LIN {X 0,Y 340.685,Z 308.673,A -85,B 0,C 180,E1 -14072.436,E2 -14072.436} C_VEL
LIN {X 0,Y 340.717,Z 308.669,A -85,B 0,C 180,E1 -14075.279,E2 -14075.279} C_VEL
LIN {X 0,Y 340.751,Z 308.84,A -85,B 0,C 180,E1 -14077.57,E2 -14077.57} C_VEL
LIN {X 0,Y 342.607,Z 316.882,A -85,B 0,C 180,E1 -14081.028,E2 -14081.028} C_VEL
LIN {X 0,Y 344.616,Z 325.417,A -85,B 0,C 180,E1 -14084.457,E2 -14084.457} C_VEL
LIN {X 0,Y 346.876,Z 334.938,A -85,B 0,C 180,E1 -14088.041,E2 -14088.041} C_VEL
LIN {X 0,Y 349.374,Z 345.213,A -85,B 0,C 180,E1 -14091.676,E2 -14091.676} C_VEL
LIN {X 0,Y 349.814,Z 347.163,A -85,B 0,C 180,E1 -14092.337,E2 -14092.337} C_VEL
LIN {X 0,Y 348.93,Z 352.343,A -85,B 0,C 180,E1 -14093.935,E2 -14093.935} C_VEL
LIN {X 0,Y 346.318,Z 365.305,A -85,B 0,C 180,E1 -14097.812,E2 -14097.812} C_VEL
LIN {X 0,Y 345.144,Z 372.439,A -85,B 0,C 180,E1 -14099.865,E2 -14099.865} C_VEL
LIN {X 0,Y 345.357,Z 374.641,A -85,B 0,C 180,E1 -14100,E2 -14100} C_VEL
LIN {X 0,Y 349.581,Z 396.16,A -85,B 0,C 180,E1 -14100.94,E2 -14100.94} C_VEL
LIN {X 0,Y 351.629,Z 411.603,A -85,B 0,C 180,E1 -14101.761,E2 -14101.761} C_VEL
LIN {X 0,Y 353.04,Z 426.596,A -85,B 0,C 180,E1 -14102.751,E2 -14102.751} C_VEL
LIN {X 0,Y 353.156,Z 435.408,A -85,B 0,C 180,E1 -14103.401,E2 -14103.401} C_VEL
LIN {X 0,Y 351.443,Z 448.562,A -85,B 0,C 180,E1 -14104.412,E2 -14104.412} C_VEL
LIN {X 0,Y 349.424,Z 461.614,A -85,B 0,C 180,E1 -14105.65,E2 -14105.65} C_VEL
LIN {X 0,Y 347.416,Z 473.933,A -85,B 0,C 180,E1 -14107.082,E2 -14107.082} C_VEL
LIN {X 0,Y 345.407,Z 486.223,A -85,B 0,C 180,E1 -14108.829,E2 -14108.829} C_VEL
LIN {X 0,Y 343.692,Z 496.83,A -85,B 0,C 180,E1 -14110.646,E2 -14110.646} C_VEL
LIN {X 0,Y 342.121,Z 506.665,A -85,B 0,C 180,E1 -14112.671,E2 -14112.671} C_VEL
LIN {X 0,Y 340.951,Z 515.073,A -85,B 0,C 180,E1 -14114.763,E2 -14114.763} C_VEL
LIN {X 0,Y 340.104,Z 522.05,A -85,B 0,C 180,E1 -14116.862,E2 -14116.862} C_VEL
LIN {X 0,Y 339.576,Z 528.54,A -85,B 0,C 180,E1 -14119.265,E2 -14119.265} C_VEL
LIN {X 0,Y 339.406,Z 533.572,A -85,B 0,C 180,E1 -14121.666,E2 -14121.666} C_VEL
LIN {X 0,Y 339.511,Z 537.273,A -85,B 0,C 180,E1 -14124.059,E2 -14124.059} C_VEL
LIN {X 0,Y 339.588,Z 539.71,A -85,B 0,C 180,E1 -14126.441,E2 -14126.441} C_VEL
LIN {X 0,Y 339.726,Z 540.943,A -85,B 0,C 180,E1 -14128.815,E2 -14128.815} C_VEL
LIN {X 0,Y 339.728,Z 540.942,A -85,B 0,C 180,E1 -14131.186,E2 -14131.186} C_VEL
LIN {X 0,Y 339.614,Z 539.708,A -85,B 0,C 180,E1 -14133.56,E2 -14133.56} C_VEL
LIN {X 0,Y 339.55,Z 537.267,A -85,B 0,C 180,E1 -14135.94,E2 -14135.94} C_VEL
LIN {X 0,Y 339.48,Z 533.556,A -85,B 0,C 180,E1 -14138.333,E2 -14138.333} C_VEL
LIN {X 0,Y 339.601,Z 528.509,A -85,B 0,C 180,E1 -14140.735,E2 -14140.735} C_VEL
LIN {X 0,Y 340.154,Z 522.02,A -85,B 0,C 180,E1 -14143.137,E2 -14143.137} C_VEL
LIN {X 0,Y 340.959,Z 515.032,A -85,B 0,C 180,E1 -14145.237,E2 -14145.237} C_VEL
LIN {X 0,Y 342.106,Z 506.607,A -85,B 0,C 180,E1 -14147.331,E2 -14147.331} C_VEL
LIN {X 0,Y 343.781,Z 496.672,A -85,B 0,C 180,E1 -14149.369,E2 -14149.369} C_VEL
LIN {X 0,Y 345.421,Z 486.141,A -85,B 0,C 180,E1 -14151.171,E2 -14151.171} C_VEL
LIN {X 0,Y 347.463,Z 473.824,A -85,B 0,C 180,E1 -14152.915,E2 -14152.915} C_VEL
LIN {X 0,Y 349.475,Z 461.488,A -85,B 0,C 180,E1 -14154.347,E2 -14154.347} C_VEL
LIN {X 0,Y 351.409,Z 448.341,A -85,B 0,C 180,E1 -14155.598,E2 -14155.598} C_VEL
LIN {X 0,Y 353.949,Z 433.264,A -85,B 0,C 180,E1 -14157.014,E2 -14157.014} C_VEL
LIN {X 0,Y 354.679,Z 418.66,A -85,B 0,C 180,E1 -14158.396,E2 -14158.396} C_VEL
LIN {X 0,Y 354.576,Z 406.998,A -85,B 0,C 180,E1 -14159.443,E2 -14159.443} C_VEL
LIN {X 0,Y 353.206,Z 394.587,A -85,B 0,C 180,E1 -14160.595,E2 -14160.595} C_VEL
LIN {X 0,Y 350.848,Z 381.951,A -85,B 0,C 180,E1 -14161.846,E2 -14161.846} C_VEL
LIN {X 0,Y 349.008,Z 374.393,A -85,B 0,C 180,E1 -14162.655,E2 -14162.655} C_VEL
LIN {X 0,Y 348.091,Z 370.111,A -85,B 0,C 180,E1 -14163.12,E2 -14163.12} C_VEL
LIN {X 0,Y 350.836,Z 361.608,A -85,B 0,C 180,E1 -14166.225,E2 -14166.225} C_VEL
LIN {X 0,Y 352.145,Z 358.36,A -85,B 0,C 180,E1 -14167.496,E2 -14167.496} C_VEL
LIN {X 0,Y 352.45,Z 356.806,A -85,B 0,C 180,E1 -14168.182,E2 -14168.182} C_VEL
LIN {X 0,Y 351.555,Z 352.589,A -85,B 0,C 180,E1 -14170.565,E2 -14170.565} C_VEL
LIN {X 0,Y 350.19,Z 348.108,A -85,B 0,C 180,E1 -14173.74,E2 -14173.74} C_VEL
LIN {X 0,Y 349.169,Z 344.785,A -85,B 0,C 180,E1 -14176.816,E2 -14176.816} C_VEL
LIN {X 0,Y 348.17,Z 342.313,A -85,B 0,C 180,E1 -14180.09,E2 -14180.09} C_VEL
LIN {X 0,Y 347.502,Z 341.045,A -85,B 0,C 180,E1 -14182.647,E2 -14182.647} C_VEL
LIN {X 0,Y 346.648,Z 340.315,A -85,B 0,C 180,E1 -14185.412,E2 -14185.412} C_VEL
LIN {X 0,Y 345.766,Z 340.093,A -85,B 0,C 180,E1 -14188.616,E2 -14188.616} C_VEL
LIN {X 0,Y 345.131,Z 340.385,A -85,B 0,C 180,E1 -14191.526,E2 -14191.526} C_VEL
LIN {X 0,Y 346.63,Z 343.275,A -85,B 0,C 180,E1 -14192.204,E2 -14192.204} C_VEL
LIN {X 0,Y 350.286,Z 348.385,A -85,B 0,C 180,E1 -14193.557,E2 -14193.557} C_VEL
LIN {X 0,Y 355.192,Z 357.489,A -85,B 0,C 180,E1 -14195.531,E2 -14195.531} C_VEL
LIN {X 0,Y 358.558,Z 365.842,A -85,B 0,C 180,E1 -14197.108,E2 -14197.108} C_VEL
LIN {X 0,Y 359.707,Z 369.419,A -85,B 0,C 180,E1 -14197.752,E2 -14197.752} C_VEL
LIN {X 0,Y 357.203,Z 382.897,A -85,B 0,C 180,E1 -14199.259,E2 -14199.259} C_VEL
LIN {X 0,Y 354.992,Z 392.974,A -85,B 0,C 180,E1 -14200.634,E2 -14200.634} C_VEL
LIN {X 0,Y 352.597,Z 403.108,A -85,B 0,C 180,E1 -14202.304,E2 -14202.304} C_VEL
LIN {X 0,Y 350.494,Z 411.648,A -85,B 0,C 180,E1 -14204.026,E2 -14204.026} C_VEL
LIN {X 0,Y 348.293,Z 419.501,A -85,B 0,C 180,E1 -14205.987,E2 -14205.987} C_VEL
LIN {X 0,Y 346.67,Z 425.084,A -85,B 0,C 180,E1 -14207.71,E2 -14207.71} C_VEL
LIN {X 0,Y 345.306,Z 429.544,A -85,B 0,C 180,E1 -14209.445,E2 -14209.445} C_VEL
LIN {X 0,Y 343.702,Z 434.016,A -85,B 0,C 180,E1 -14211.771,E2 -14211.771} C_VEL
LIN {X 0,Y 343.116,Z 435.597,A -85,B 0,C 180,E1 -14212.941,E2 -14212.941} C_VEL
LIN {X 0,Y 342.313,Z 437.544,A -85,B 0,C 180,E1 -14215.289,E2 -14215.289} C_VEL
LIN {X 0,Y 341.557,Z 438.025,A -85,B 0,C 180,E1 -14217.642,E2 -14217.642} C_VEL
LIN {X 0,Y 341.362,Z 437.648,A -85,B 0,C 180,E1 -14218.82,E2 -14218.82} C_VEL
LIN {X 0,Y 341.018,Z 436.906,A -85,B 0,C 180,E1 -14220,E2 -14220} C_VEL
LIN {X 0,Y 340.978,Z 435.738,A -85,B 0,C 180,E1 -14221.181,E2 -14221.181} C_VEL
LIN {X 0,Y 340.851,Z 434.198,A -85,B 0,C 180,E1 -14222.364,E2 -14222.364} C_VEL
LIN {X 0,Y 340.813,Z 431.07,A -85,B 0,C 180,E1 -14224.139,E2 -14224.139} C_VEL
LIN {X 0,Y 341.181,Z 426.928,A -85,B 0,C 180,E1 -14225.912,E2 -14225.912} C_VEL
LIN {X 0,Y 341.536,Z 421.737,A -85,B 0,C 180,E1 -14227.687,E2 -14227.687} C_VEL
LIN {X 0,Y 342.068,Z 414.154,A -85,B 0,C 180,E1 -14229.759,E2 -14229.759} C_VEL
LIN {X 0,Y 342.657,Z 406.099,A -85,B 0,C 180,E1 -14231.536,E2 -14231.536} C_VEL
LIN {X 0,Y 343.362,Z 396.351,A -85,B 0,C 180,E1 -14233.313,E2 -14233.313} C_VEL
LIN {X 0,Y 344.291,Z 385.473,A -85,B 0,C 180,E1 -14234.935,E2 -14234.935} C_VEL
LIN {X 0,Y 345.287,Z 373.449,A -85,B 0,C 180,E1 -14236.404,E2 -14236.404} C_VEL
LIN {X 0,Y 346.141,Z 361.256,A -85,B 0,C 180,E1 -14237.624,E2 -14237.624} C_VEL
LIN {X 0,Y 346.99,Z 348.049,A -85,B 0,C 180,E1 -14238.679,E2 -14238.679} C_VEL
LIN {X 0,Y 343.823,Z 334.91,A -85,B 0,C 180,E1 -14239.681,E2 -14239.681} C_VEL
LIN {X 0,Y 340.174,Z 320.362,A -85,B 0,C 180,E1 -14240.562,E2 -14240.562} C_VEL
LIN {X 0,Y 340.178,Z 316.024,A -85,B 0,C 180,E1 -14244.627,E2 -14244.627} C_VEL
LIN {X 0,Y 340.19,Z 312.178,A -85,B 0,C 180,E1 -14248.37,E2 -14248.37} C_VEL
LIN {X 0,Y 340.199,Z 309.423,A -85,B 0,C 180,E1 -14251.095,E2 -14251.095} C_VEL
LIN {X 0,Y 340.306,Z 308.722,A -85,B 0,C 180,E1 -14252.477,E2 -14252.477} C_VEL
LIN {X 0,Y 340.556,Z 308.69,A -85,B 0,C 180,E1 -14255.298,E2 -14255.298} C_VEL
LIN {X 0,Y 340.705,Z 308.671,A -85,B 0,C 180,E1 -14258.384,E2 -14258.384} C_VEL
LIN {X 0,Y 340.701,Z 308.665,A -85,B 0,C 180,E1 -14262.045,E2 -14262.045} C_VEL
LIN {X 0,Y 340.707,Z 308.817,A -85,B 0,C 180,E1 -14263.132,E2 -14263.132} C_VEL
LIN {X 0,Y 341.39,Z 312.413,A -85,B 0,C 180,E1 -14266.098,E2 -14266.098} C_VEL
LIN {X 0,Y 341.716,Z 315.809,A -85,B 0,C 180,E1 -14268.842,E2 -14268.842} C_VEL
LIN {X 0,Y 341.73,Z 319.739,A -85,B 0,C 180,E1 -14271.904,E2 -14271.904} C_VEL
LIN {X 0,Y 341.66,Z 324.36,A -85,B 0,C 180,E1 -14275.367,E2 -14275.367} C_VEL
LIN {X 0,Y 341.617,Z 329.636,A -85,B 0,C 180,E1 -14279.048,E2 -14279.048} C_VEL
LIN {X 0,Y 341.643,Z 330.583,A -85,B 0,C 180,E1 -14279.625,E2 -14279.625} C_VEL
LIN {X 0,Y 343.082,Z 333.899,A -85,B 0,C 180,E1 -14279.849,E2 -14279.849} C_VEL
LIN {X 0,Y 349.127,Z 348.085,A -85,B 0,C 180,E1 -14280.902,E2 -14280.902} C_VEL
LIN {X 0,Y 354.05,Z 362.001,A -85,B 0,C 180,E1 -14282.041,E2 -14282.041} C_VEL
LIN {X 0,Y 356.741,Z 371.631,A -85,B 0,C 180,E1 -14282.881,E2 -14282.881} C_VEL
LIN {X 0,Y 355.481,Z 385.325,A -85,B 0,C 180,E1 -14283.838,E2 -14283.838} C_VEL
LIN {X 0,Y 353.788,Z 399.027,A -85,B 0,C 180,E1 -14285.03,E2 -14285.03} C_VEL
LIN {X 0,Y 351.753,Z 412.252,A -85,B 0,C 180,E1 -14286.447,E2 -14286.447} C_VEL
LIN {X 0,Y 349.877,Z 424.229,A -85,B 0,C 180,E1 -14288.03,E2 -14288.03} C_VEL
LIN {X 0,Y 347.873,Z 435.957,A -85,B 0,C 180,E1 -14289.913,E2 -14289.913} C_VEL
LIN {X 0,Y 346.162,Z 445.017,A -85,B 0,C 180,E1 -14291.658,E2 -14291.658} C_VEL
LIN {X 0,Y 344.321,Z 454.308,A -85,B 0,C 180,E1 -14293.804,E2 -14293.804} C_VEL
LIN {X 0,Y 343.032,Z 461.257,A -85,B 0,C 180,E1 -14295.767,E2 -14295.767} C_VEL
LIN {X 0,Y 341.82,Z 468.102,A -85,B 0,C 180,E1 -14298.135,E2 -14298.135} C_VEL
LIN {X 0,Y 340.917,Z 473.474,A -85,B 0,C 180,E1 -14300.507,E2 -14300.507} C_VEL
LIN {X 0,Y 340.273,Z 477.532,A -85,B 0,C 180,E1 -14302.881,E2 -14302.881} C_VEL
LIN {X 0,Y 340.001,Z 480.366,A -85,B 0,C 180,E1 -14305.257,E2 -14305.257} C_VEL
LIN {X 0,Y 339.76,Z 482.072,A -85,B 0,C 180,E1 -14307.629,E2 -14307.629} C_VEL
LIN {X 0,Y 339.624,Z 482.668,A -85,B 0,C 180,E1 -14310,E2 -14310} C_VEL
LIN {X 0,Y 339.755,Z 482.11,A -85,B 0,C 180,E1 -14312.371,E2 -14312.371} C_VEL
LIN {X 0,Y 339.998,Z 480.455,A -85,B 0,C 180,E1 -14314.743,E2 -14314.743} C_VEL
LIN {X 0,Y 340.272,Z 477.68,A -85,B 0,C 180,E1 -14317.118,E2 -14317.118} C_VEL
LIN {X 0,Y 340.909,Z 473.685,A -85,B 0,C 180,E1 -14319.493,E2 -14319.493} C_VEL
LIN {X 0,Y 341.793,Z 468.373,A -85,B 0,C 180,E1 -14321.866,E2 -14321.866} C_VEL
LIN {X 0,Y 343.01,Z 461.588,A -85,B 0,C 180,E1 -14324.233,E2 -14324.233} C_VEL
LIN {X 0,Y 344.226,Z 454.918,A -85,B 0,C 180,E1 -14326.142,E2 -14326.142} C_VEL
LIN {X 0,Y 346.053,Z 445.516,A -85,B 0,C 180,E1 -14328.348,E2 -14328.348} C_VEL
LIN {X 0,Y 348.106,Z 434.858,A -85,B 0,C 180,E1 -14330.381,E2 -14330.381} C_VEL
LIN {X 0,Y 349.849,Z 423.919,A -85,B 0,C 180,E1 -14332.127,E2 -14332.127} C_VEL
LIN {X 0,Y 351.938,Z 411.859,A -85,B 0,C 180,E1 -14333.696,E2 -14333.696} C_VEL
LIN {X 0,Y 353.85,Z 398.537,A -85,B 0,C 180,E1 -14335.121,E2 -14335.121} C_VEL
LIN {X 0,Y 355.533,Z 384.643,A -85,B 0,C 180,E1 -14336.32,E2 -14336.32} C_VEL
LIN {X 0,Y 356.766,Z 372.504,A -85,B 0,C 180,E1 -14337.161,E2 -14337.161} C_VEL
LIN {X 0,Y 355.958,Z 368.246,A -85,B 0,C 180,E1 -14337.515,E2 -14337.515} C_VEL
LIN {X 0,Y 351.475,Z 354.305,A -85,B 0,C 180,E1 -14338.709,E2 -14338.709} C_VEL
LIN {X 0,Y 345.813,Z 339.855,A -85,B 0,C 180,E1 -14339.821,E2 -14339.821} C_VEL
LIN {X 0,Y 341.718,Z 330.796,A -85,B 0,C 180,E1 -14340.473,E2 -14340.473} C_VEL
LIN {X 0,Y 341.639,Z 330.42,A -85,B 0,C 180,E1 -14340.544,E2 -14340.544} C_VEL
LIN {X 0,Y 341.624,Z 325.783,A -85,B 0,C 180,E1 -14343.742,E2 -14343.742} C_VEL
LIN {X 0,Y 341.659,Z 322.309,A -85,B 0,C 180,E1 -14346.3,E2 -14346.3} C_VEL
LIN {X 0,Y 341.072,Z 321.186,A -85,B 0,C 180,E1 -14347.266,E2 -14347.266} C_VEL
LIN {X 0,Y 338.315,Z 319.77,A -85,B 0,C 180,E1 -14348.851,E2 -14348.851} C_VEL
LIN {X 0,Y 335.921,Z 318.68,A -85,B 0,C 180,E1 -14350.136,E2 -14350.136} C_VEL
LIN {X 0,Y 334.857,Z 317.669,A -85,B 0,C 180,E1 -14351.124,E2 -14351.124} C_VEL
LIN {X 0,Y 334.753,Z 317.262,A -85,B 0,C 180,E1 -14351.456,E2 -14351.456} C_VEL
LIN {X 0,Y 334.404,Z 313.699,A -85,B 0,C 180,E1 -14354.393,E2 -14354.393} C_VEL
LIN {X 0,Y 333.652,Z 309.552,A -85,B 0,C 180,E1 -14357.824,E2 -14357.824} C_VEL
LIN {X 0,Y 333.652,Z 309.545,A -85,B 0,C 180,E1 -14361.202,E2 -14361.202} C_VEL
LIN {X 0,Y 333.676,Z 309.541,A -85,B 0,C 180,E1 -14363.861,E2 -14363.861} C_VEL
LIN {X 0,Y 333.643,Z 309.547,A -85,B 0,C 180,E1 -14367.413,E2 -14367.413} C_VEL
LIN {X 0,Y 333.652,Z 309.545,A -85,B 0,C 180,E1 -14371.022,E2 -14371.022} C_VEL
LIN {X 0,Y 333.694,Z 309.538,A -85,B 0,C 180,E1 -14375.088,E2 -14375.088} C_VEL
LIN {X 0,Y 333.673,Z 309.535,A -85,B 0,C 180,E1 -14379.019,E2 -14379.019} C_VEL
LIN {X 0,Y 333.741,Z 309.534,A -85,B 0,C 180,E1 -14381.586,E2 -14381.586} C_VEL
LIN {X 0,Y 333.808,Z 309.531,A -85,B 0,C 180,E1 -14385.577,E2 -14385.577} C_VEL
LIN {X 0,Y 333.817,Z 309.513,A -85,B 0,C 180,E1 -14389.077,E2 -14389.077} C_VEL
LIN {X 0,Y 333.957,Z 309.5,A -85,B 0,C 180,E1 -14392.746,E2 -14392.746} C_VEL
LIN {X 0,Y 333.796,Z 309.519,A -85,B 0,C 180,E1 -14395.169,E2 -14395.169} C_VEL
LIN {X 0,Y 334.103,Z 309.49,A -85,B 0,C 180,E1 -14397.589,E2 -14397.589} C_VEL
LIN {X 0,Y 334.227,Z 309.456,A -85,B 0,C 180,E1 -14400,E2 -14400} C_VEL
LIN {X 0,Y 334.092,Z 309.494,A -85,B 0,C 180,E1 -14402.411,E2 -14402.411} C_VEL
LIN {X 0,Y 334.001,Z 309.488,A -85,B 0,C 180,E1 -14406.039,E2 -14406.039} C_VEL
LIN {X 0,Y 333.82,Z 309.517,A -85,B 0,C 180,E1 -14409.696,E2 -14409.696} C_VEL
LIN {X 0,Y 333.797,Z 309.531,A -85,B 0,C 180,E1 -14413.391,E2 -14413.391} C_VEL
LIN {X 0,Y 333.745,Z 309.521,A -85,B 0,C 180,E1 -14417.146,E2 -14417.146} C_VEL
LIN {X 0,Y 333.731,Z 309.54,A -85,B 0,C 180,E1 -14419.691,E2 -14419.691} C_VEL
LIN {X 0,Y 333.659,Z 309.547,A -85,B 0,C 180,E1 -14423.591,E2 -14423.591} C_VEL
LIN {X 0,Y 333.656,Z 309.533,A -85,B 0,C 180,E1 -14426.253,E2 -14426.253} C_VEL
LIN {X 0,Y 333.661,Z 309.549,A -85,B 0,C 180,E1 -14430.278,E2 -14430.278} C_VEL
LIN {X 0,Y 333.636,Z 309.551,A -85,B 0,C 180,E1 -14433.208,E2 -14433.208} C_VEL
LIN {X 0,Y 333.665,Z 309.548,A -85,B 0,C 180,E1 -14436.832,E2 -14436.832} C_VEL
LIN {X 0,Y 335.573,Z 317.725,A -85,B 0,C 180,E1 -14440.484,E2 -14440.484} C_VEL
LIN {X 0,Y 337.662,Z 326.748,A -85,B 0,C 180,E1 -14444.207,E2 -14444.207} C_VEL
LIN {X 0,Y 340.037,Z 336.8,A -85,B 0,C 180,E1 -14448.078,E2 -14448.078} C_VEL
LIN {X 0,Y 342.687,Z 347.803,A -85,B 0,C 180,E1 -14452.03,E2 -14452.03} C_VEL
LIN {X 0,Y 342.709,Z 349.82,A -85,B 0,C 180,E1 -14452.693,E2 -14452.693} C_VEL
LIN {X 0,Y 340.309,Z 360.87,A -85,B 0,C 180,E1 -14456.11,E2 -14456.11} C_VEL
LIN {X 0,Y 338.556,Z 370.259,A -85,B 0,C 180,E1 -14458.967,E2 -14458.967} C_VEL
LIN {X 0,Y 338.549,Z 372.627,A -85,B 0,C 180,E1 -14459.297,E2 -14459.297} C_VEL
LIN {X 0,Y 343.01,Z 395.522,A -85,B 0,C 180,E1 -14460.325,E2 -14460.325} C_VEL
LIN {X 0,Y 345.131,Z 410.993,A -85,B 0,C 180,E1 -14461.179,E2 -14461.179} C_VEL
LIN {X 0,Y 346.5,Z 425.999,A -85,B 0,C 180,E1 -14462.193,E2 -14462.193} C_VEL
LIN {X 0,Y 346.519,Z 436.8,A -85,B 0,C 180,E1 -14463.012,E2 -14463.012} C_VEL
LIN {X 0,Y 344.46,Z 451.393,A -85,B 0,C 180,E1 -14464.205,E2 -14464.205} C_VEL
LIN {X 0,Y 342.263,Z 464.914,A -85,B 0,C 180,E1 -14465.591,E2 -14465.591} C_VEL
LIN {X 0,Y 340.232,Z 476.565,A -85,B 0,C 180,E1 -14467.053,E2 -14467.053} C_VEL
LIN {X 0,Y 338.395,Z 487.419,A -85,B 0,C 180,E1 -14468.688,E2 -14468.688} C_VEL
LIN {X 0,Y 336.674,Z 497.471,A -85,B 0,C 180,E1 -14470.489,E2 -14470.489} C_VEL
LIN {X 0,Y 335.028,Z 507.311,A -85,B 0,C 180,E1 -14472.607,E2 -14472.607} C_VEL
LIN {X 0,Y 333.858,Z 515.529,A -85,B 0,C 180,E1 -14474.744,E2 -14474.744} C_VEL
LIN {X 0,Y 332.913,Z 523.208,A -85,B 0,C 180,E1 -14477.194,E2 -14477.194} C_VEL
LIN {X 0,Y 332.448,Z 529.329,A -85,B 0,C 180,E1 -14479.648,E2 -14479.648} C_VEL
LIN {X 0,Y 332.337,Z 534.039,A -85,B 0,C 180,E1 -14482.1,E2 -14482.1} C_VEL
LIN {X 0,Y 332.427,Z 536.661,A -85,B 0,C 180,E1 -14483.932,E2 -14483.932} C_VEL
LIN {X 0,Y 332.493,Z 539.099,A -85,B 0,C 180,E1 -14486.365,E2 -14486.365} C_VEL
LIN {X 0,Y 332.646,Z 540.334,A -85,B 0,C 180,E1 -14488.79,E2 -14488.79} C_VEL
LIN {X 0,Y 332.664,Z 540.335,A -85,B 0,C 180,E1 -14491.211,E2 -14491.211} C_VEL
LIN {X 0,Y 332.52,Z 539.097,A -85,B 0,C 180,E1 -14493.636,E2 -14493.636} C_VEL
LIN {X 0,Y 332.462,Z 536.098,A -85,B 0,C 180,E1 -14496.515,E2 -14496.515} C_VEL
LIN {X 0,Y 332.402,Z 531.831,A -85,B 0,C 180,E1 -14499.124,E2 -14499.124} C_VEL
LIN {X 0,Y 332.701,Z 526.426,A -85,B 0,C 180,E1 -14501.577,E2 -14501.577} C_VEL
LIN {X 0,Y 333.406,Z 519.179,A -85,B 0,C 180,E1 -14504.152,E2 -14504.152} C_VEL
LIN {X 0,Y 334.466,Z 510.985,A -85,B 0,C 180,E1 -14506.48,E2 -14506.48} C_VEL
LIN {X 0,Y 335.976,Z 501.867,A -85,B 0,C 180,E1 -14508.603,E2 -14508.603} C_VEL
LIN {X 0,Y 337.571,Z 492.271,A -85,B 0,C 180,E1 -14510.468,E2 -14510.468} C_VEL
LIN {X 0,Y 339.437,Z 481.628,A -85,B 0,C 180,E1 -14512.202,E2 -14512.202} C_VEL
LIN {X 0,Y 341.391,Z 469.678,A -85,B 0,C 180,E1 -14513.829,E2 -14513.829} C_VEL
LIN {X 0,Y 343.649,Z 456.65,A -85,B 0,C 180,E1 -14515.272,E2 -14515.272} C_VEL
LIN {X 0,Y 345.111,Z 447.959,A -85,B 0,C 180,E1 -14516.164,E2 -14516.164} C_VEL
LIN {X 0,Y 347.779,Z 434.682,A -85,B 0,C 180,E1 -14517.533,E2 -14517.533} C_VEL
LIN {X 0,Y 348.841,Z 418.132,A -85,B 0,C 180,E1 -14519.179,E2 -14519.179} C_VEL
LIN {X 0,Y 348.722,Z 405.794,A -85,B 0,C 180,E1 -14520.359,E2 -14520.359} C_VEL
LIN {X 0,Y 347.14,Z 391.953,A -85,B 0,C 180,E1 -14521.762,E2 -14521.762} C_VEL
LIN {X 0,Y 344.518,Z 378.598,A -85,B 0,C 180,E1 -14523.24,E2 -14523.24} C_VEL
LIN {X 0,Y 342.958,Z 372.452,A -85,B 0,C 180,E1 -14523.998,E2 -14523.998} C_VEL
LIN {X 0,Y 342.265,Z 368.564,A -85,B 0,C 180,E1 -14524.471,E2 -14524.471} C_VEL
LIN {X 0,Y 345.314,Z 360.419,A -85,B 0,C 180,E1 -14527.632,E2 -14527.632} C_VEL
LIN {X 0,Y 345.694,Z 358.877,A -85,B 0,C 180,E1 -14528.322,E2 -14528.322} C_VEL
LIN {X 0,Y 344.673,Z 354.258,A -85,B 0,C 180,E1 -14531.024,E2 -14531.024} C_VEL
LIN {X 0,Y 343.335,Z 349.933,A -85,B 0,C 180,E1 -14534.239,E2 -14534.239} C_VEL
LIN {X 0,Y 342.306,Z 346.748,A -85,B 0,C 180,E1 -14537.349,E2 -14537.349} C_VEL
LIN {X 0,Y 341.421,Z 344.552,A -85,B 0,C 180,E1 -14540.348,E2 -14540.348} C_VEL
LIN {X 0,Y 340.598,Z 343.194,A -85,B 0,C 180,E1 -14543.245,E2 -14543.245} C_VEL
LIN {X 0,Y 339.751,Z 342.508,A -85,B 0,C 180,E1 -14546.047,E2 -14546.047} C_VEL
LIN {X 0,Y 338.704,Z 342.416,A -85,B 0,C 180,E1 -14549.918,E2 -14549.918} C_VEL
LIN {X 0,Y 340.182,Z 345.183,A -85,B 0,C 180,E1 -14550.692,E2 -14550.692} C_VEL
LIN {X 0,Y 341.572,Z 346.471,A -85,B 0,C 180,E1 -14551.235,E2 -14551.235} C_VEL
LIN {X 0,Y 342.864,Z 348.93,A -85,B 0,C 180,E1 -14551.872,E2 -14551.872} C_VEL
LIN {X 0,Y 346.193,Z 354.01,A -85,B 0,C 180,E1 -14553.283,E2 -14553.283} C_VEL
LIN {X 0,Y 350.159,Z 361.747,A -85,B 0,C 180,E1 -14555.072,E2 -14555.072} C_VEL
LIN {X 0,Y 353.302,Z 370.051,A -85,B 0,C 180,E1 -14556.748,E2 -14556.748} C_VEL
LIN {X 0,Y 353.826,Z 371.673,A -85,B 0,C 180,E1 -14557.061,E2 -14557.061} C_VEL
LIN {X 0,Y 353.934,Z 373.412,A -85,B 0,C 180,E1 -14557.318,E2 -14557.318} C_VEL
LIN {X 0,Y 351.324,Z 385.499,A -85,B 0,C 180,E1 -14558.742,E2 -14558.742} C_VEL
LIN {X 0,Y 348.807,Z 396.193,A -85,B 0,C 180,E1 -14560.276,E2 -14560.276} C_VEL
LIN {X 0,Y 346.268,Z 405.931,A -85,B 0,C 180,E1 -14561.97,E2 -14561.97} C_VEL
LIN {X 0,Y 343.773,Z 414.942,A -85,B 0,C 180,E1 -14563.917,E2 -14563.917} C_VEL
LIN {X 0,Y 341.736,Z 421.72,A -85,B 0,C 180,E1 -14565.713,E2 -14565.713} C_VEL
LIN {X 0,Y 340.009,Z 427.039,A -85,B 0,C 180,E1 -14567.465,E2 -14567.465} C_VEL
LIN {X 0,Y 338.57,Z 431.354,A -85,B 0,C 180,E1 -14569.233,E2 -14569.233} C_VEL
LIN {X 0,Y 337.706,Z 433.699,A -85,B 0,C 180,E1 -14570.416,E2 -14570.416} C_VEL
LIN {X 0,Y 336.882,Z 435.607,A -85,B 0,C 180,E1 -14571.603,E2 -14571.603} C_VEL
LIN {X 0,Y 335.748,Z 438.167,A -85,B 0,C 180,E1 -14573.992,E2 -14573.992} C_VEL
LIN {X 0,Y 335.389,Z 438.879,A -85,B 0,C 180,E1 -14575.192,E2 -14575.192} C_VEL
LIN {X 0,Y 334.959,Z 439.237,A -85,B 0,C 180,E1 -14576.391,E2 -14576.391} C_VEL
LIN {X 0,Y 334.567,Z 439.186,A -85,B 0,C 180,E1 -14577.592,E2 -14577.592} C_VEL
LIN {X 0,Y 334.36,Z 438.724,A -85,B 0,C 180,E1 -14578.796,E2 -14578.796} C_VEL
LIN {X 0,Y 333.99,Z 437.912,A -85,B 0,C 180,E1 -14580,E2 -14580} C_VEL
LIN {X 0,Y 333.952,Z 436.677,A -85,B 0,C 180,E1 -14581.206,E2 -14581.206} C_VEL
LIN {X 0,Y 333.731,Z 434.07,A -85,B 0,C 180,E1 -14583.018,E2 -14583.018} C_VEL
LIN {X 0,Y 333.828,Z 430.489,A -85,B 0,C 180,E1 -14584.831,E2 -14584.831} C_VEL
LIN {X 0,Y 334.297,Z 425.875,A -85,B 0,C 180,E1 -14586.64,E2 -14586.64} C_VEL
LIN {X 0,Y 334.706,Z 419.182,A -85,B 0,C 180,E1 -14588.738,E2 -14588.738} C_VEL
LIN {X 0,Y 335.213,Z 411.922,A -85,B 0,C 180,E1 -14590.571,E2 -14590.571} C_VEL
LIN {X 0,Y 335.921,Z 403.185,A -85,B 0,C 180,E1 -14592.383,E2 -14592.383} C_VEL
LIN {X 0,Y 336.752,Z 392.58,A -85,B 0,C 180,E1 -14594.195,E2 -14594.195} C_VEL
LIN {X 0,Y 337.723,Z 381.842,A -85,B 0,C 180,E1 -14595.696,E2 -14595.696} C_VEL
LIN {X 0,Y 338.797,Z 368.632,A -85,B 0,C 180,E1 -14597.209,E2 -14597.209} C_VEL
LIN {X 0,Y 339.658,Z 355.761,A -85,B 0,C 180,E1 -14598.394,E2 -14598.394} C_VEL
LIN {X 0,Y 339.997,Z 348.981,A -85,B 0,C 180,E1 -14598.922,E2 -14598.922} C_VEL
LIN {X 0,Y 336.609,Z 334.812,A -85,B 0,C 180,E1 -14600.023,E2 -14600.023} C_VEL
LIN {X 0,Y 333.128,Z 320.921,A -85,B 0,C 180,E1 -14600.898,E2 -14600.898} C_VEL
LIN {X 0,Y 333.122,Z 316.621,A -85,B 0,C 180,E1 -14604.958,E2 -14604.958} C_VEL
LIN {X 0,Y 333.171,Z 313.855,A -85,B 0,C 180,E1 -14607.65,E2 -14607.65} C_VEL
LIN {X 0,Y 333.172,Z 311.068,A -85,B 0,C 180,E1 -14610.415,E2 -14610.415} C_VEL
LIN {X 0,Y 333.183,Z 309.68,A -85,B 0,C 180,E1 -14611.826,E2 -14611.826} C_VEL
LIN {X 0,Y 333.47,Z 309.567,A -85,B 0,C 180,E1 -14614.72,E2 -14614.72} C_VEL
LIN {X 0,Y 333.638,Z 309.55,A -85,B 0,C 180,E1 -14617.653,E2 -14617.653} C_VEL
LIN {X 0,Y 333.652,Z 309.543,A -85,B 0,C 180,E1 -14621.568,E2 -14621.568} C_VEL
LIN {X 0,Y 333.666,Z 309.785,A -85,B 0,C 180,E1 -14622.506,E2 -14622.506} C_VEL
LIN {X 0,Y 334.482,Z 314.069,A -85,B 0,C 180,E1 -14626.101,E2 -14626.101} C_VEL
LIN {X 0,Y 334.818,Z 317.727,A -85,B 0,C 180,E1 -14629.083,E2 -14629.083} C_VEL
LIN {X 0,Y 334.758,Z 322.132,A -85,B 0,C 180,E1 -14632.494,E2 -14632.494} C_VEL
LIN {X 0,Y 334.707,Z 327.128,A -85,B 0,C 180,E1 -14636.19,E2 -14636.19} C_VEL
LIN {X 0,Y 334.715,Z 331.069,A -85,B 0,C 180,E1 -14638.909,E2 -14638.909} C_VEL
LIN {X 0,Y 336.087,Z 334.342,A -85,B 0,C 180,E1 -14639.15,E2 -14639.15} C_VEL
LIN {X 0,Y 342.256,Z 348.54,A -85,B 0,C 180,E1 -14640.253,E2 -14640.253} C_VEL
LIN {X 0,Y 347.138,Z 362.138,A -85,B 0,C 180,E1 -14641.405,E2 -14641.405} C_VEL
LIN {X 0,Y 350.25,Z 372.598,A -85,B 0,C 180,E1 -14642.362,E2 -14642.362} C_VEL
LIN {X 0,Y 349.118,Z 386.217,A -85,B 0,C 180,E1 -14643.349,E2 -14643.349} C_VEL
LIN {X 0,Y 347.392,Z 399.624,A -85,B 0,C 180,E1 -14644.538,E2 -14644.538} C_VEL
LIN {X 0,Y 345.304,Z 412.85,A -85,B 0,C 180,E1 -14645.979,E2 -14645.979} C_VEL
LIN {X 0,Y 343.329,Z 424.832,A -85,B 0,C 180,E1 -14647.588,E2 -14647.588} C_VEL
LIN {X 0,Y 341.228,Z 436.563,A -85,B 0,C 180,E1 -14649.504,E2 -14649.504} C_VEL
LIN {X 0,Y 339.434,Z 445.626,A -85,B 0,C 180,E1 -14651.281,E2 -14651.281} C_VEL
LIN {X 0,Y 337.48,Z 455.146,A -85,B 0,C 180,E1 -14653.527,E2 -14653.527} C_VEL
LIN {X 0,Y 336.16,Z 461.867,A -85,B 0,C 180,E1 -14655.47,E2 -14655.47} C_VEL
LIN {X 0,Y 334.897,Z 468.711,A -85,B 0,C 180,E1 -14657.886,E2 -14657.886} C_VEL
LIN {X 0,Y 333.921,Z 474.084,A -85,B 0,C 180,E1 -14660.306,E2 -14660.306} C_VEL
LIN {X 0,Y 333.252,Z 478.141,A -85,B 0,C 180,E1 -14662.73,E2 -14662.73} C_VEL
LIN {X 0,Y 332.94,Z 480.976,A -85,B 0,C 180,E1 -14665.156,E2 -14665.156} C_VEL
LIN {X 0,Y 332.696,Z 482.68,A -85,B 0,C 180,E1 -14667.578,E2 -14667.578} C_VEL
LIN {X 0,Y 332.565,Z 483.275,A -85,B 0,C 180,E1 -14670,E2 -14670} C_VEL
LIN {X 0,Y 332.691,Z 482.718,A -85,B 0,C 180,E1 -14672.421,E2 -14672.421} C_VEL
LIN {X 0,Y 332.937,Z 481.064,A -85,B 0,C 180,E1 -14674.843,E2 -14674.843} C_VEL
LIN {X 0,Y 333.252,Z 478.287,A -85,B 0,C 180,E1 -14677.269,E2 -14677.269} C_VEL
LIN {X 0,Y 333.91,Z 474.294,A -85,B 0,C 180,E1 -14679.693,E2 -14679.693} C_VEL
LIN {X 0,Y 334.869,Z 468.979,A -85,B 0,C 180,E1 -14682.115,E2 -14682.115} C_VEL
LIN {X 0,Y 336.137,Z 462.194,A -85,B 0,C 180,E1 -14684.53,E2 -14684.53} C_VEL
LIN {X 0,Y 337.63,Z 454.425,A -85,B 0,C 180,E1 -14686.76,E2 -14686.76} C_VEL
LIN {X 0,Y 339.338,Z 446.118,A -85,B 0,C 180,E1 -14688.724,E2 -14688.724} C_VEL
LIN {X 0,Y 341.481,Z 435.457,A -85,B 0,C 180,E1 -14690.795,E2 -14690.795} C_VEL
LIN {X 0,Y 343.295,Z 424.516,A -85,B 0,C 180,E1 -14692.572,E2 -14692.572} C_VEL
LIN {X 0,Y 345.472,Z 412.45,A -85,B 0,C 180,E1 -14694.167,E2 -14694.167} C_VEL
LIN {X 0,Y 347.467,Z 399.122,A -85,B 0,C 180,E1 -14695.616,E2 -14695.616} C_VEL
LIN {X 0,Y 349.177,Z 385.613,A -85,B 0,C 180,E1 -14696.804,E2 -14696.804} C_VEL
LIN {X 0,Y 350.38,Z 373.196,A -85,B 0,C 180,E1 -14697.69,E2 -14697.69} C_VEL
LIN {X 0,Y 346.258,Z 359.276,A -85,B 0,C 180,E1 -14698.954,E2 -14698.954} C_VEL
LIN {X 0,Y 340.948,Z 345.189,A -85,B 0,C 180,E1 -14700.123,E2 -14700.123} C_VEL
LIN {X 0,Y 335.692,Z 333.707,A -85,B 0,C 180,E1 -14701.02,E2 -14701.02} C_VEL
LIN {X 0,Y 334.733,Z 331.08,A -85,B 0,C 180,E1 -14701.208,E2 -14701.208} C_VEL
LIN {X 0,Y 334.72,Z 325.633,A -85,B 0,C 180,E1 -14705.028,E2 -14705.028} C_VEL
LIN {X 0,Y 334.805,Z 321.329,A -85,B 0,C 180,E1 -14708.261,E2 -14708.261} C_VEL
LIN {X 0,Y 334.753,Z 317.262,A -85,B 0,C 180,E1 -14711.456,E2 -14711.456} C_VEL
LIN {X 0,Y 334.002,Z 316.199,A -85,B 0,C 180,E1 -14712.442,E2 -14712.442} C_VEL
LIN {X 0,Y 330.961,Z 314.947,A -85,B 0,C 180,E1 -14714.054,E2 -14714.054} C_VEL
LIN {X 0,Y 328.343,Z 313.933,A -85,B 0,C 180,E1 -14715.361,E2 -14715.361} C_VEL
LIN {X 0,Y 327.125,Z 312.975,A -85,B 0,C 180,E1 -14716.372,E2 -14716.372} C_VEL
LIN {X 0,Y 326.974,Z 312.6,A -85,B 0,C 180,E1 -14716.714,E2 -14716.714} C_VEL
LIN {X 0,Y 326.602,Z 310.424,A -85,B 0,C 180,E1 -14718.785,E2 -14718.785} C_VEL
LIN {X 0,Y 326.627,Z 310.422,A -85,B 0,C 180,E1 -14722.761,E2 -14722.761} C_VEL
LIN {X 0,Y 326.607,Z 310.42,A -85,B 0,C 180,E1 -14725.98,E2 -14725.98} C_VEL
LIN {X 0,Y 326.611,Z 310.418,A -85,B 0,C 180,E1 -14729.397,E2 -14729.397} C_VEL
LIN {X 0,Y 326.607,Z 310.417,A -85,B 0,C 180,E1 -14733.135,E2 -14733.135} C_VEL
LIN {X 0,Y 326.632,Z 310.425,A -85,B 0,C 180,E1 -14735.869,E2 -14735.869} C_VEL
LIN {X 0,Y 326.65,Z 310.418,A -85,B 0,C 180,E1 -14739.864,E2 -14739.864} C_VEL
LIN {X 0,Y 326.664,Z 310.405,A -85,B 0,C 180,E1 -14742.47,E2 -14742.47} C_VEL
LIN {X 0,Y 326.759,Z 310.408,A -85,B 0,C 180,E1 -14746.314,E2 -14746.314} C_VEL
LIN {X 0,Y 326.783,Z 310.399,A -85,B 0,C 180,E1 -14750.093,E2 -14750.093} C_VEL
LIN {X 0,Y 326.944,Z 310.364,A -85,B 0,C 180,E1 -14753.83,E2 -14753.83} C_VEL
LIN {X 0,Y 327.044,Z 310.37,A -85,B 0,C 180,E1 -14757.537,E2 -14757.537} C_VEL
LIN {X 0,Y 327.179,Z 310.334,A -85,B 0,C 180,E1 -14760,E2 -14760} C_VEL
LIN {X 0,Y 327.033,Z 310.374,A -85,B 0,C 180,E1 -14762.463,E2 -14762.463} C_VEL
LIN {X 0,Y 326.957,Z 310.366,A -85,B 0,C 180,E1 -14766.17,E2 -14766.17} C_VEL
LIN {X 0,Y 326.783,Z 310.39,A -85,B 0,C 180,E1 -14769.907,E2 -14769.907} C_VEL
LIN {X 0,Y 326.759,Z 310.41,A -85,B 0,C 180,E1 -14773.685,E2 -14773.685} C_VEL
LIN {X 0,Y 326.698,Z 310.403,A -85,B 0,C 180,E1 -14777.528,E2 -14777.528} C_VEL
LIN {X 0,Y 326.657,Z 310.415,A -85,B 0,C 180,E1 -14780.135,E2 -14780.135} C_VEL
LIN {X 0,Y 326.632,Z 310.425,A -85,B 0,C 180,E1 -14784.13,E2 -14784.13} C_VEL
LIN {X 0,Y 326.601,Z 310.424,A -85,B 0,C 180,E1 -14788.084,E2 -14788.084} C_VEL
LIN {X 0,Y 326.573,Z 310.431,A -85,B 0,C 180,E1 -14791.097,E2 -14791.097} C_VEL
LIN {X 0,Y 326.606,Z 310.426,A -85,B 0,C 180,E1 -14794.019,E2 -14794.019} C_VEL
LIN {X 0,Y 326.642,Z 310.553,A -85,B 0,C 180,E1 -14796.277,E2 -14796.277} C_VEL
LIN {X 0,Y 328.519,Z 318.538,A -85,B 0,C 180,E1 -14799.925,E2 -14799.925} C_VEL
LIN {X 0,Y 330.551,Z 327.461,A -85,B 0,C 180,E1 -14803.707,E2 -14803.707} C_VEL
LIN {X 0,Y 332.782,Z 336.987,A -85,B 0,C 180,E1 -14807.483,E2 -14807.483} C_VEL
LIN {X 0,Y 335.29,Z 347.362,A -85,B 0,C 180,E1 -14811.332,E2 -14811.332} C_VEL
LIN {X 0,Y 335.832,Z 349.949,A -85,B 0,C 180,E1 -14812.257,E2 -14812.257} C_VEL
LIN {X 0,Y 334.243,Z 357.435,A -85,B 0,C 180,E1 -14814.651,E2 -14814.651} C_VEL
LIN {X 0,Y 331.943,Z 368.472,A -85,B 0,C 180,E1 -14818.083,E2 -14818.083} C_VEL
LIN {X 0,Y 332.008,Z 372.148,A -85,B 0,C 180,E1 -14818.625,E2 -14818.625} C_VEL
LIN {X 0,Y 336.501,Z 395.138,A -85,B 0,C 180,E1 -14819.699,E2 -14819.699} C_VEL
LIN {X 0,Y 338.61,Z 410.662,A -85,B 0,C 180,E1 -14820.584,E2 -14820.584} C_VEL
LIN {X 0,Y 339.892,Z 425.393,A -85,B 0,C 180,E1 -14821.603,E2 -14821.603} C_VEL
LIN {X 0,Y 340.086,Z 436.209,A -85,B 0,C 180,E1 -14822.459,E2 -14822.459} C_VEL
LIN {X 0,Y 338.19,Z 450.029,A -85,B 0,C 180,E1 -14823.61,E2 -14823.61} C_VEL
LIN {X 0,Y 335.976,Z 463.014,A -85,B 0,C 180,E1 -14824.939,E2 -14824.939} C_VEL
LIN {X 0,Y 333.6,Z 475.957,A -85,B 0,C 180,E1 -14826.569,E2 -14826.569} C_VEL
LIN {X 0,Y 331.681,Z 486.808,A -85,B 0,C 180,E1 -14828.235,E2 -14828.235} C_VEL
LIN {X 0,Y 329.907,Z 496.86,A -85,B 0,C 180,E1 -14830.072,E2 -14830.072} C_VEL
LIN {X 0,Y 328.168,Z 506.698,A -85,B 0,C 180,E1 -14832.231,E2 -14832.231} C_VEL
LIN {X 0,Y 326.911,Z 514.913,A -85,B 0,C 180,E1 -14834.412,E2 -14834.412} C_VEL
LIN {X 0,Y 325.9,Z 522.592,A -85,B 0,C 180,E1 -14836.913,E2 -14836.913} C_VEL
LIN {X 0,Y 325.394,Z 528.714,A -85,B 0,C 180,E1 -14839.422,E2 -14839.422} C_VEL
LIN {X 0,Y 325.234,Z 533.423,A -85,B 0,C 180,E1 -14841.926,E2 -14841.926} C_VEL
LIN {X 0,Y 325.368,Z 536.051,A -85,B 0,C 180,E1 -14843.8,E2 -14843.8} C_VEL
LIN {X 0,Y 325.401,Z 538.488,A -85,B 0,C 180,E1 -14846.285,E2 -14846.285} C_VEL
LIN {X 0,Y 325.57,Z 539.725,A -85,B 0,C 180,E1 -14848.763,E2 -14848.763} C_VEL
LIN {X 0,Y 325.587,Z 539.726,A -85,B 0,C 180,E1 -14851.237,E2 -14851.237} C_VEL
LIN {X 0,Y 325.429,Z 538.486,A -85,B 0,C 180,E1 -14853.715,E2 -14853.715} C_VEL
LIN {X 0,Y 325.375,Z 535.682,A -85,B 0,C 180,E1 -14856.495,E2 -14856.495} C_VEL
LIN {X 0,Y 325.314,Z 532.324,A -85,B 0,C 180,E1 -14858.698,E2 -14858.698} C_VEL
LIN {X 0,Y 325.505,Z 527.275,A -85,B 0,C 180,E1 -14861.205,E2 -14861.205} C_VEL
LIN {X 0,Y 326.113,Z 520.78,A -85,B 0,C 180,E1 -14863.713,E2 -14863.713} C_VEL
LIN {X 0,Y 327.206,Z 512.651,A -85,B 0,C 180,E1 -14866.214,E2 -14866.214} C_VEL
LIN {X 0,Y 328.659,Z 504.005,A -85,B 0,C 180,E1 -14868.386,E2 -14868.386} C_VEL
LIN {X 0,Y 330.519,Z 493.633,A -85,B 0,C 180,E1 -14870.536,E2 -14870.536} C_VEL
LIN {X 0,Y 332.418,Z 482.987,A -85,B 0,C 180,E1 -14872.369,E2 -14872.369} C_VEL
LIN {X 0,Y 334.425,Z 471.434,A -85,B 0,C 180,E1 -14874.027,E2 -14874.027} C_VEL
LIN {X 0,Y 336.712,Z 458.91,A -85,B 0,C 180,E1 -14875.499,E2 -14875.499} C_VEL
LIN {X 0,Y 337.846,Z 453.066,A -85,B 0,C 180,E1 -14876.173,E2 -14876.173} C_VEL
LIN {X 0,Y 341.15,Z 438.827,A -85,B 0,C 180,E1 -14877.781,E2 -14877.781} C_VEL
LIN {X 0,Y 342.626,Z 425.993,A -85,B 0,C 180,E1 -14879.155,E2 -14879.155} C_VEL
LIN {X 0,Y 343.224,Z 410.983,A -85,B 0,C 180,E1 -14880.682,E2 -14880.682} C_VEL
LIN {X 0,Y 342.325,Z 397.821,A -85,B 0,C 180,E1 -14882.089,E2 -14882.089} C_VEL
LIN {X 0,Y 340.061,Z 382.91,A -85,B 0,C 180,E1 -14883.811,E2 -14883.811} C_VEL
LIN {X 0,Y 337.68,Z 372.092,A -85,B 0,C 180,E1 -14885.236,E2 -14885.236} C_VEL
LIN {X 0,Y 336.674,Z 367.457,A -85,B 0,C 180,E1 -14885.883,E2 -14885.883} C_VEL
LIN {X 0,Y 336.668,Z 366.972,A -85,B 0,C 180,E1 -14885.953,E2 -14885.953} C_VEL
LIN {X 0,Y 338.66,Z 362.075,A -85,B 0,C 180,E1 -14887.946,E2 -14887.946} C_VEL
LIN {X 0,Y 338.942,Z 360.953,A -85,B 0,C 180,E1 -14888.467,E2 -14888.467} C_VEL
LIN {X 0,Y 338.09,Z 357.03,A -85,B 0,C 180,E1 -14890.783,E2 -14890.783} C_VEL
LIN {X 0,Y 336.941,Z 353.278,A -85,B 0,C 180,E1 -14893.498,E2 -14893.498} C_VEL
LIN {X 0,Y 335.967,Z 350.112,A -85,B 0,C 180,E1 -14896.345,E2 -14896.345} C_VEL
LIN {X 0,Y 334.987,Z 347.569,A -85,B 0,C 180,E1 -14899.43,E2 -14899.43} C_VEL
LIN {X 0,Y 334.155,Z 345.894,A -85,B 0,C 180,E1 -14902.416,E2 -14902.416} C_VEL
LIN {X 0,Y 333.232,Z 344.963,A -85,B 0,C 180,E1 -14905.339,E2 -14905.339} C_VEL
LIN {X 0,Y 332.485,Z 344.779,A -85,B 0,C 180,E1 -14908.055,E2 -14908.055} C_VEL
LIN {X 0,Y 333.622,Z 346.987,A -85,B 0,C 180,E1 -14908.807,E2 -14908.807} C_VEL
LIN {X 0,Y 335.676,Z 349.369,A -85,B 0,C 180,E1 -14909.836,E2 -14909.836} C_VEL
LIN {X 0,Y 336.784,Z 351.245,A -85,B 0,C 180,E1 -14910.455,E2 -14910.455} C_VEL
LIN {X 0,Y 337.83,Z 352.271,A -85,B 0,C 180,E1 -14910.897,E2 -14910.897} C_VEL
LIN {X 0,Y 343.129,Z 361.617,A -85,B 0,C 180,E1 -14913.542,E2 -14913.542} C_VEL
LIN {X 0,Y 346.099,Z 368.295,A -85,B 0,C 180,E1 -14915.125,E2 -14915.125} C_VEL
LIN {X 0,Y 348.346,Z 375.198,A -85,B 0,C 180,E1 -14916.568,E2 -14916.568} C_VEL
LIN {X 0,Y 348.025,Z 377.771,A -85,B 0,C 180,E1 -14916.911,E2 -14916.911} C_VEL
LIN {X 0,Y 344.997,Z 390.332,A -85,B 0,C 180,E1 -14918.489,E2 -14918.489} C_VEL
LIN {X 0,Y 342.174,Z 401.08,A -85,B 0,C 180,E1 -14920.19,E2 -14920.19} C_VEL
LIN {X 0,Y 339.575,Z 410.15,A -85,B 0,C 180,E1 -14921.914,E2 -14921.914} C_VEL
LIN {X 0,Y 337.271,Z 417.681,A -85,B 0,C 180,E1 -14923.662,E2 -14923.662} C_VEL
LIN {X 0,Y 334.568,Z 425.758,A -85,B 0,C 180,E1 -14926.021,E2 -14926.021} C_VEL
LIN {X 0,Y 332.838,Z 430.546,A -85,B 0,C 180,E1 -14927.81,E2 -14927.81} C_VEL
LIN {X 0,Y 331.369,Z 434.307,A -85,B 0,C 180,E1 -14929.614,E2 -14929.614} C_VEL
LIN {X 0,Y 330.05,Z 437.205,A -85,B 0,C 180,E1 -14931.428,E2 -14931.428} C_VEL
LIN {X 0,Y 328.839,Z 439.604,A -85,B 0,C 180,E1 -14933.866,E2 -14933.866} C_VEL
LIN {X 0,Y 328.458,Z 440.217,A -85,B 0,C 180,E1 -14935.09,E2 -14935.09} C_VEL
LIN {X 0,Y 327.574,Z 440.334,A -85,B 0,C 180,E1 -14937.541,E2 -14937.541} C_VEL
LIN {X 0,Y 327.354,Z 439.8,A -85,B 0,C 180,E1 -14938.77,E2 -14938.77} C_VEL
LIN {X 0,Y 326.963,Z 438.915,A -85,B 0,C 180,E1 -14940,E2 -14940} C_VEL
LIN {X 0,Y 326.925,Z 437.598,A -85,B 0,C 180,E1 -14941.232,E2 -14941.232} C_VEL
LIN {X 0,Y 326.697,Z 434.872,A -85,B 0,C 180,E1 -14943.083,E2 -14943.083} C_VEL
LIN {X 0,Y 326.805,Z 431.163,A -85,B 0,C 180,E1 -14944.935,E2 -14944.935} C_VEL
LIN {X 0,Y 327.256,Z 426.412,A -85,B 0,C 180,E1 -14946.783,E2 -14946.783} C_VEL
LIN {X 0,Y 327.614,Z 420.561,A -85,B 0,C 180,E1 -14948.637,E2 -14948.637} C_VEL
LIN {X 0,Y 328.142,Z 413.438,A -85,B 0,C 180,E1 -14950.489,E2 -14950.489} C_VEL
LIN {X 0,Y 328.848,Z 404.796,A -85,B 0,C 180,E1 -14952.34,E2 -14952.34} C_VEL
LIN {X 0,Y 329.668,Z 394.326,A -85,B 0,C 180,E1 -14954.192,E2 -14954.192} C_VEL
LIN {X 0,Y 330.765,Z 382.646,A -85,B 0,C 180,E1 -14955.877,E2 -14955.877} C_VEL
LIN {X 0,Y 331.857,Z 369.32,A -85,B 0,C 180,E1 -14957.44,E2 -14957.44} C_VEL
LIN {X 0,Y 332.724,Z 356.746,A -85,B 0,C 180,E1 -14958.626,E2 -14958.626} C_VEL
LIN {X 0,Y 333.102,Z 350.264,A -85,B 0,C 180,E1 -14959.143,E2 -14959.143} C_VEL
LIN {X 0,Y 330.06,Z 337.41,A -85,B 0,C 180,E1 -14960.182,E2 -14960.182} C_VEL
LIN {X 0,Y 326.372,Z 322.854,A -85,B 0,C 180,E1 -14961.121,E2 -14961.121} C_VEL
LIN {X 0,Y 326.071,Z 321.511,A -85,B 0,C 180,E1 -14961.21,E2 -14961.21} C_VEL
LIN {X 0,Y 326.063,Z 316.961,A -85,B 0,C 180,E1 -14965.536,E2 -14965.536} C_VEL
LIN {X 0,Y 326.108,Z 314.15,A -85,B 0,C 180,E1 -14968.303,E2 -14968.303} C_VEL
LIN {X 0,Y 326.135,Z 311.316,A -85,B 0,C 180,E1 -14971.144,E2 -14971.144} C_VEL
LIN {X 0,Y 326.231,Z 310.476,A -85,B 0,C 180,E1 -14972.84,E2 -14972.84} C_VEL
LIN {X 0,Y 326.477,Z 310.445,A -85,B 0,C 180,E1 -14975.537,E2 -14975.537} C_VEL
LIN {X 0,Y 326.595,Z 310.427,A -85,B 0,C 180,E1 -14978.613,E2 -14978.613} C_VEL
LIN {X 0,Y 326.624,Z 310.499,A -85,B 0,C 180,E1 -14981.636,E2 -14981.636} C_VEL
LIN {X 0,Y 327.37,Z 314.558,A -85,B 0,C 180,E1 -14985.109,E2 -14985.109} C_VEL
LIN {X 0,Y 327.699,Z 316.633,A -85,B 0,C 180,E1 -14986.818,E2 -14986.818} C_VEL
LIN {X 0,Y 327.896,Z 320.542,A -85,B 0,C 180,E1 -14989.983,E2 -14989.983} C_VEL
LIN {X 0,Y 327.848,Z 324.615,A -85,B 0,C 180,E1 -14993.113,E2 -14993.113} C_VEL
LIN {X 0,Y 327.79,Z 329.579,A -85,B 0,C 180,E1 -14996.739,E2 -14996.739} C_VEL
LIN {X 0,Y 327.862,Z 331.87,A -85,B 0,C 180,E1 -14998.206,E2 -14998.206} C_VEL
LIN {X 0,Y 330.471,Z 337.768,A -85,B 0,C 180,E1 -14998.648,E2 -14998.648} C_VEL
LIN {X 0,Y 336.124,Z 350.735,A -85,B 0,C 180,E1 -14999.721,E2 -14999.721} C_VEL
LIN {X 0,Y 341.084,Z 364.679,A -85,B 0,C 180,E1 -15000.964,E2 -15000.964} C_VEL
LIN {X 0,Y 343.955,Z 375.226,A -85,B 0,C 180,E1 -15001.968,E2 -15001.968} C_VEL
LIN {X 0,Y 342.469,Z 389.495,A -85,B 0,C 180,E1 -15003.046,E2 -15003.046} C_VEL
LIN {X 0,Y 340.588,Z 403.034,A -85,B 0,C 180,E1 -15004.32,E2 -15004.32} C_VEL
LIN {X 0,Y 338.437,Z 415.721,A -85,B 0,C 180,E1 -15005.783,E2 -15005.783} C_VEL
LIN {X 0,Y 336.613,Z 426.404,A -85,B 0,C 180,E1 -15007.278,E2 -15007.278} C_VEL
LIN {X 0,Y 334.612,Z 437.168,A -85,B 0,C 180,E1 -15009.08,E2 -15009.08} C_VEL
LIN {X 0,Y 332.724,Z 446.233,A -85,B 0,C 180,E1 -15010.889,E2 -15010.889} C_VEL
LIN {X 0,Y 330.901,Z 454.644,A -85,B 0,C 180,E1 -15012.893,E2 -15012.893} C_VEL
LIN {X 0,Y 329.298,Z 462.477,A -85,B 0,C 180,E1 -15015.16,E2 -15015.16} C_VEL
LIN {X 0,Y 327.983,Z 469.319,A -85,B 0,C 180,E1 -15017.626,E2 -15017.626} C_VEL
LIN {X 0,Y 326.929,Z 474.695,A -85,B 0,C 180,E1 -15020.097,E2 -15020.097} C_VEL
LIN {X 0,Y 326.226,Z 478.751,A -85,B 0,C 180,E1 -15022.573,E2 -15022.573} C_VEL
LIN {X 0,Y 325.883,Z 481.585,A -85,B 0,C 180,E1 -15025.051,E2 -15025.051} C_VEL
LIN {X 0,Y 325.634,Z 483.288,A -85,B 0,C 180,E1 -15027.526,E2 -15027.526} C_VEL
LIN {X 0,Y 325.492,Z 483.883,A -85,B 0,C 180,E1 -15030,E2 -15030} C_VEL
LIN {X 0,Y 325.629,Z 483.325,A -85,B 0,C 180,E1 -15032.474,E2 -15032.474} C_VEL
LIN {X 0,Y 325.88,Z 481.672,A -85,B 0,C 180,E1 -15034.948,E2 -15034.948} C_VEL
LIN {X 0,Y 326.227,Z 478.895,A -85,B 0,C 180,E1 -15037.427,E2 -15037.427} C_VEL
LIN {X 0,Y 326.917,Z 474.902,A -85,B 0,C 180,E1 -15039.903,E2 -15039.903} C_VEL
LIN {X 0,Y 327.956,Z 469.584,A -85,B 0,C 180,E1 -15042.374,E2 -15042.374} C_VEL
LIN {X 0,Y 329.274,Z 462.8,A -85,B 0,C 180,E1 -15044.84,E2 -15044.84} C_VEL
LIN {X 0,Y 330.821,Z 455.227,A -85,B 0,C 180,E1 -15047.062,E2 -15047.062} C_VEL
LIN {X 0,Y 332.647,Z 446.719,A -85,B 0,C 180,E1 -15049.115,E2 -15049.115} C_VEL
LIN {X 0,Y 334.876,Z 436.056,A -85,B 0,C 180,E1 -15051.224,E2 -15051.224} C_VEL
LIN {X 0,Y 336.758,Z 425.113,A -85,B 0,C 180,E1 -15053.035,E2 -15053.035} C_VEL
LIN {X 0,Y 339.025,Z 413.043,A -85,B 0,C 180,E1 -15054.657,E2 -15054.657} C_VEL
LIN {X 0,Y 341.1,Z 399.709,A -85,B 0,C 180,E1 -15056.13,E2 -15056.13} C_VEL
LIN {X 0,Y 342.837,Z 386.576,A -85,B 0,C 180,E1 -15057.308,E2 -15057.308} C_VEL
LIN {X 0,Y 344.068,Z 375.211,A -85,B 0,C 180,E1 -15058.132,E2 -15058.132} C_VEL
LIN {X 0,Y 340.106,Z 361.676,A -85,B 0,C 180,E1 -15059.42,E2 -15059.42} C_VEL
LIN {X 0,Y 334.918,Z 347.647,A -85,B 0,C 180,E1 -15060.643,E2 -15060.643} C_VEL
LIN {X 0,Y 327.993,Z 332.254,A -85,B 0,C 180,E1 -15061.884,E2 -15061.884} C_VEL
LIN {X 0,Y 327.86,Z 331.682,A -85,B 0,C 180,E1 -15061.944,E2 -15061.944} C_VEL
LIN {X 0,Y 327.813,Z 326.737,A -85,B 0,C 180,E1 -15065.444,E2 -15065.444} C_VEL
LIN {X 0,Y 327.918,Z 322.787,A -85,B 0,C 180,E1 -15068.428,E2 -15068.428} C_VEL
LIN {X 0,Y 327.839,Z 318.709,A -85,B 0,C 180,E1 -15071.648,E2 -15071.648} C_VEL
LIN {X 0,Y 327.642,Z 316.613,A -85,B 0,C 180,E1 -15073.346,E2 -15073.346} C_VEL
LIN {X 0,Y 326.974,Z 312.6,A -85,B 0,C 180,E1 -15076.714,E2 -15076.714} C_VEL
LIN {X 0,Y 326.135,Z 311.713,A -85,B 0,C 180,E1 -15077.726,E2 -15077.726} C_VEL
LIN {X 0,Y 323.13,Z 311.177,A -85,B 0,C 180,E1 -15079.39,E2 -15079.39} C_VEL
LIN {X 0,Y 320.68,Z 311.217,A -85,B 0,C 180,E1 -15080.747,E2 -15080.747} C_VEL
LIN {X 0,Y 319.651,Z 311.297,A -85,B 0,C 180,E1 -15081.798,E2 -15081.798} C_VEL
LIN {X 0,Y 319.573,Z 311.304,A -85,B 0,C 180,E1 -15082.154,E2 -15082.154} C_VEL
LIN {X 0,Y 319.561,Z 311.307,A -85,B 0,C 180,E1 -15085.123,E2 -15085.123} C_VEL
LIN {X 0,Y 319.524,Z 311.31,A -85,B 0,C 180,E1 -15088.137,E2 -15088.137} C_VEL
LIN {X 0,Y 319.569,Z 311.304,A -85,B 0,C 180,E1 -15091.604,E2 -15091.604} C_VEL
LIN {X 0,Y 319.573,Z 311.299,A -85,B 0,C 180,E1 -15095.301,E2 -15095.301} C_VEL
LIN {X 0,Y 319.567,Z 311.288,A -85,B 0,C 180,E1 -15098.045,E2 -15098.045} C_VEL
LIN {X 0,Y 319.657,Z 311.292,A -85,B 0,C 180,E1 -15100.979,E2 -15100.979} C_VEL
LIN {X 0,Y 319.712,Z 311.285,A -85,B 0,C 180,E1 -15105.289,E2 -15105.289} C_VEL
LIN {X 0,Y 319.715,Z 311.266,A -85,B 0,C 180,E1 -15108.589,E2 -15108.589} C_VEL
LIN {X 0,Y 319.853,Z 311.261,A -85,B 0,C 180,E1 -15112.424,E2 -15112.424} C_VEL
LIN {X 0,Y 319.731,Z 311.268,A -85,B 0,C 180,E1 -15114.956,E2 -15114.956} C_VEL
LIN {X 0,Y 319.987,Z 311.249,A -85,B 0,C 180,E1 -15117.482,E2 -15117.482} C_VEL
LIN {X 0,Y 320.132,Z 311.211,A -85,B 0,C 180,E1 -15120,E2 -15120} C_VEL
LIN {X 0,Y 319.976,Z 311.253,A -85,B 0,C 180,E1 -15122.518,E2 -15122.518} C_VEL
LIN {X 0,Y 319.914,Z 311.244,A -85,B 0,C 180,E1 -15126.306,E2 -15126.306} C_VEL
LIN {X 0,Y 319.735,Z 311.265,A -85,B 0,C 180,E1 -15130.128,E2 -15130.128} C_VEL
LIN {X 0,Y 319.732,Z 311.283,A -85,B 0,C 180,E1 -15133.992,E2 -15133.992} C_VEL
LIN {X 0,Y 319.658,Z 311.285,A -85,B 0,C 180,E1 -15137.927,E2 -15137.927} C_VEL
LIN {X 0,Y 319.601,Z 311.288,A -85,B 0,C 180,E1 -15140.6,E2 -15140.6} C_VEL
LIN {X 0,Y 319.573,Z 311.303,A -85,B 0,C 180,E1 -15144.698,E2 -15144.698} C_VEL
LIN {X 0,Y 319.57,Z 311.302,A -85,B 0,C 180,E1 -15148.396,E2 -15148.396} C_VEL
LIN {X 0,Y 319.523,Z 311.31,A -85,B 0,C 180,E1 -15151.863,E2 -15151.863} C_VEL
LIN {X 0,Y 319.582,Z 311.399,A -85,B 0,C 180,E1 -15155.61,E2 -15155.61} C_VEL
LIN {X 0,Y 321.437,Z 319.352,A -85,B 0,C 180,E1 -15159.351,E2 -15159.351} C_VEL
LIN {X 0,Y 323.436,Z 328.155,A -85,B 0,C 180,E1 -15163.194,E2 -15163.194} C_VEL
LIN {X 0,Y 325.724,Z 337.952,A -85,B 0,C 180,E1 -15167.189,E2 -15167.189} C_VEL
LIN {X 0,Y 328.174,Z 348.189,A -85,B 0,C 180,E1 -15171.09,E2 -15171.09} C_VEL
LIN {X 0,Y 328.796,Z 351.434,A -85,B 0,C 180,E1 -15172.267,E2 -15172.267} C_VEL
LIN {X 0,Y 326.617,Z 360.852,A -85,B 0,C 180,E1 -15175.342,E2 -15175.342} C_VEL
LIN {X 0,Y 325.481,Z 366.357,A -85,B 0,C 180,E1 -15177.099,E2 -15177.099} C_VEL
LIN {X 0,Y 325.44,Z 371.762,A -85,B 0,C 180,E1 -15177.92,E2 -15177.92} C_VEL
LIN {X 0,Y 329.327,Z 390.656,A -85,B 0,C 180,E1 -15178.834,E2 -15178.834} C_VEL
LIN {X 0,Y 331.494,Z 405.118,A -85,B 0,C 180,E1 -15179.638,E2 -15179.638} C_VEL
LIN {X 0,Y 332.958,Z 419.65,A -85,B 0,C 180,E1 -15180.608,E2 -15180.608} C_VEL
LIN {X 0,Y 333.615,Z 432.595,A -85,B 0,C 180,E1 -15181.621,E2 -15181.621} C_VEL
LIN {X 0,Y 333.286,Z 439.472,A -85,B 0,C 180,E1 -15182.19,E2 -15182.19} C_VEL
LIN {X 0,Y 331.156,Z 453.175,A -85,B 0,C 180,E1 -15183.416,E2 -15183.416} C_VEL
LIN {X 0,Y 328.804,Z 466.241,A -85,B 0,C 180,E1 -15184.861,E2 -15184.861} C_VEL
LIN {X 0,Y 326.451,Z 478.532,A -85,B 0,C 180,E1 -15186.53,E2 -15186.53} C_VEL
LIN {X 0,Y 324.345,Z 489.775,A -85,B 0,C 180,E1 -15188.386,E2 -15188.386} C_VEL
LIN {X 0,Y 322.324,Z 500.703,A -85,B 0,C 180,E1 -15190.579,E2 -15190.579} C_VEL
LIN {X 0,Y 320.659,Z 509.801,A -85,B 0,C 180,E1 -15192.79,E2 -15192.79} C_VEL
LIN {X 0,Y 319.371,Z 518.343,A -85,B 0,C 180,E1 -15195.341,E2 -15195.341} C_VEL
LIN {X 0,Y 318.569,Z 525.222,A -85,B 0,C 180,E1 -15197.902,E2 -15197.902} C_VEL
LIN {X 0,Y 318.185,Z 530.62,A -85,B 0,C 180,E1 -15200.465,E2 -15200.465} C_VEL
LIN {X 0,Y 318.18,Z 533.743,A -85,B 0,C 180,E1 -15202.385,E2 -15202.385} C_VEL
LIN {X 0,Y 318.293,Z 535.44,A -85,B 0,C 180,E1 -15203.662,E2 -15203.662} C_VEL
LIN {X 0,Y 318.31,Z 537.877,A -85,B 0,C 180,E1 -15206.202,E2 -15206.202} C_VEL
LIN {X 0,Y 318.459,Z 538.651,A -85,B 0,C 180,E1 -15207.471,E2 -15207.471} C_VEL
LIN {X 0,Y 318.555,Z 539.281,A -85,B 0,C 180,E1 -15210,E2 -15210} C_VEL
LIN {X 0,Y 318.479,Z 538.65,A -85,B 0,C 180,E1 -15212.53,E2 -15212.53} C_VEL
LIN {X 0,Y 318.307,Z 536.805,A -85,B 0,C 180,E1 -15215.067,E2 -15215.067} C_VEL
LIN {X 0,Y 318.219,Z 533.727,A -85,B 0,C 180,E1 -15217.615,E2 -15217.615} C_VEL
LIN {X 0,Y 318.282,Z 529.353,A -85,B 0,C 180,E1 -15220.175,E2 -15220.175} C_VEL
LIN {X 0,Y 318.725,Z 523.599,A -85,B 0,C 180,E1 -15222.739,E2 -15222.739} C_VEL
LIN {X 0,Y 319.675,Z 516.318,A -85,B 0,C 180,E1 -15225.297,E2 -15225.297} C_VEL
LIN {X 0,Y 320.824,Z 508.528,A -85,B 0,C 180,E1 -15227.531,E2 -15227.531} C_VEL
LIN {X 0,Y 322.619,Z 499.189,A -85,B 0,C 180,E1 -15229.734,E2 -15229.734} C_VEL
LIN {X 0,Y 324.377,Z 489.69,A -85,B 0,C 180,E1 -15231.613,E2 -15231.613} C_VEL
LIN {X 0,Y 326.715,Z 477.393,A -85,B 0,C 180,E1 -15233.619,E2 -15233.619} C_VEL
LIN {X 0,Y 328.774,Z 466.097,A -85,B 0,C 180,E1 -15235.142,E2 -15235.142} C_VEL
LIN {X 0,Y 330.298,Z 458.857,A -85,B 0,C 180,E1 -15236.031,E2 -15236.031} C_VEL
LIN {X 0,Y 333.389,Z 446.497,A -85,B 0,C 180,E1 -15237.631,E2 -15237.631} C_VEL
LIN {X 0,Y 335.523,Z 437.544,A -85,B 0,C 180,E1 -15238.63,E2 -15238.63} C_VEL
LIN {X 0,Y 337.167,Z 422.586,A -85,B 0,C 180,E1 -15240.306,E2 -15240.306} C_VEL
LIN {X 0,Y 337.658,Z 409.996,A -85,B 0,C 180,E1 -15241.673,E2 -15241.673} C_VEL
LIN {X 0,Y 336.625,Z 395.457,A -85,B 0,C 180,E1 -15243.373,E2 -15243.373} C_VEL
LIN {X 0,Y 334.713,Z 382.538,A -85,B 0,C 180,E1 -15245.027,E2 -15245.027} C_VEL
LIN {X 0,Y 333.276,Z 375.358,A -85,B 0,C 180,E1 -15246.069,E2 -15246.069} C_VEL
LIN {X 0,Y 332.379,Z 370.779,A -85,B 0,C 180,E1 -15246.759,E2 -15246.759} C_VEL
LIN {X 0,Y 331.413,Z 366.413,A -85,B 0,C 180,E1 -15247.471,E2 -15247.471} C_VEL
LIN {X 0,Y 331.387,Z 365.155,A -85,B 0,C 180,E1 -15247.666,E2 -15247.666} C_VEL
LIN {X 0,Y 332.106,Z 363.351,A -85,B 0,C 180,E1 -15248.465,E2 -15248.465} C_VEL
LIN {X 0,Y 331.624,Z 360.22,A -85,B 0,C 180,E1 -15250.277,E2 -15250.277} C_VEL
LIN {X 0,Y 330.209,Z 355.534,A -85,B 0,C 180,E1 -15253.644,E2 -15253.644} C_VEL
LIN {X 0,Y 329.138,Z 352.032,A -85,B 0,C 180,E1 -15256.899,E2 -15256.899} C_VEL
LIN {X 0,Y 328.014,Z 349.324,A -85,B 0,C 180,E1 -15260.474,E2 -15260.474} C_VEL
LIN {X 0,Y 327.293,Z 348.033,A -85,B 0,C 180,E1 -15263.041,E2 -15263.041} C_VEL
LIN {X 0,Y 326.433,Z 347.345,A -85,B 0,C 180,E1 -15265.673,E2 -15265.673} C_VEL
LIN {X 0,Y 327.679,Z 349.656,A -85,B 0,C 180,E1 -15266.769,E2 -15266.769} C_VEL
LIN {X 0,Y 329.34,Z 351.003,A -85,B 0,C 180,E1 -15267.758,E2 -15267.758} C_VEL
LIN {X 0,Y 330.977,Z 353.738,A -85,B 0,C 180,E1 -15268.85,E2 -15268.85} C_VEL
LIN {X 0,Y 334.072,Z 358.086,A -85,B 0,C 180,E1 -15270.603,E2 -15270.603} C_VEL
LIN {X 0,Y 338.62,Z 366.672,A -85,B 0,C 180,E1 -15273.184,E2 -15273.184} C_VEL
LIN {X 0,Y 341.44,Z 373.634,A -85,B 0,C 180,E1 -15274.914,E2 -15274.914} C_VEL
LIN {X 0,Y 342.957,Z 378.89,A -85,B 0,C 180,E1 -15276.095,E2 -15276.095} C_VEL
LIN {X 0,Y 339.762,Z 391.133,A -85,B 0,C 180,E1 -15277.661,E2 -15277.661} C_VEL
LIN {X 0,Y 336.486,Z 402.715,A -85,B 0,C 180,E1 -15279.522,E2 -15279.522} C_VEL
LIN {X 0,Y 333.697,Z 411.62,A -85,B 0,C 180,E1 -15281.266,E2 -15281.266} C_VEL
LIN {X 0,Y 330.935,Z 419.889,A -85,B 0,C 180,E1 -15283.258,E2 -15283.258} C_VEL
LIN {X 0,Y 328.667,Z 426.168,A -85,B 0,C 180,E1 -15285.132,E2 -15285.132} C_VEL
LIN {X 0,Y 326.181,Z 432.52,A -85,B 0,C 180,E1 -15287.557,E2 -15287.557} C_VEL
LIN {X 0,Y 324.631,Z 436.121,A -85,B 0,C 180,E1 -15289.396,E2 -15289.396} C_VEL
LIN {X 0,Y 323.237,Z 438.806,A -85,B 0,C 180,E1 -15291.246,E2 -15291.246} C_VEL
LIN {X 0,Y 321.949,Z 441.035,A -85,B 0,C 180,E1 -15293.734,E2 -15293.734} C_VEL
LIN {X 0,Y 321.52,Z 441.539,A -85,B 0,C 180,E1 -15294.984,E2 -15294.984} C_VEL
LIN {X 0,Y 320.578,Z 441.479,A -85,B 0,C 180,E1 -15297.487,E2 -15297.487} C_VEL
LIN {X 0,Y 320.346,Z 440.863,A -85,B 0,C 180,E1 -15298.743,E2 -15298.743} C_VEL
LIN {X 0,Y 319.933,Z 439.904,A -85,B 0,C 180,E1 -15300,E2 -15300} C_VEL
LIN {X 0,Y 319.899,Z 438.474,A -85,B 0,C 180,E1 -15301.259,E2 -15301.259} C_VEL
LIN {X 0,Y 319.662,Z 435.629,A -85,B 0,C 180,E1 -15303.151,E2 -15303.151} C_VEL
LIN {X 0,Y 319.784,Z 431.794,A -85,B 0,C 180,E1 -15305.043,E2 -15305.043} C_VEL
LIN {X 0,Y 320.221,Z 426.923,A -85,B 0,C 180,E1 -15306.933,E2 -15306.933} C_VEL
LIN {X 0,Y 320.706,Z 419.45,A -85,B 0,C 180,E1 -15309.237,E2 -15309.237} C_VEL
LIN {X 0,Y 321.377,Z 410.874,A -85,B 0,C 180,E1 -15311.351,E2 -15311.351} C_VEL
LIN {X 0,Y 322.103,Z 401.464,A -85,B 0,C 180,E1 -15313.244,E2 -15313.244} C_VEL
LIN {X 0,Y 323.165,Z 390.028,A -85,B 0,C 180,E1 -15315.128,E2 -15315.128} C_VEL
LIN {X 0,Y 324.202,Z 378.425,A -85,B 0,C 180,E1 -15316.692,E2 -15316.692} C_VEL
LIN {X 0,Y 325.2,Z 365.518,A -85,B 0,C 180,E1 -15318.12,E2 -15318.12} C_VEL
LIN {X 0,Y 326.177,Z 352.608,A -85,B 0,C 180,E1 -15319.267,E2 -15319.267} C_VEL
LIN {X 0,Y 324.501,Z 344.176,A -85,B 0,C 180,E1 -15319.987,E2 -15319.987} C_VEL
LIN {X 0,Y 321.066,Z 330.214,A -85,B 0,C 180,E1 -15321.019,E2 -15321.019} C_VEL
LIN {X 0,Y 319.03,Z 322.11,A -85,B 0,C 180,E1 -15321.528,E2 -15321.528} C_VEL
LIN {X 0,Y 319.042,Z 318.032,A -85,B 0,C 180,E1 -15325.422,E2 -15325.422} C_VEL
LIN {X 0,Y 319.078,Z 314.437,A -85,B 0,C 180,E1 -15328.985,E2 -15328.985} C_VEL
LIN {X 0,Y 319.108,Z 311.554,A -85,B 0,C 180,E1 -15331.909,E2 -15331.909} C_VEL
LIN {X 0,Y 319.452,Z 311.32,A -85,B 0,C 180,E1 -15335.51,E2 -15335.51} C_VEL
LIN {X 0,Y 319.532,Z 311.307,A -85,B 0,C 180,E1 -15338.014,E2 -15338.014} C_VEL
LIN {X 0,Y 319.585,Z 311.452,A -85,B 0,C 180,E1 -15340.861,E2 -15340.861} C_VEL
LIN {X 0,Y 320.383,Z 315.719,A -85,B 0,C 180,E1 -15344.585,E2 -15344.585} C_VEL
LIN {X 0,Y 320.84,Z 318.871,A -85,B 0,C 180,E1 -15347.23,E2 -15347.23} C_VEL
LIN {X 0,Y 320.984,Z 323.023,A -85,B 0,C 180,E1 -15350.582,E2 -15350.582} C_VEL
LIN {X 0,Y 320.917,Z 327.684,A -85,B 0,C 180,E1 -15354.125,E2 -15354.125} C_VEL
LIN {X 0,Y 320.898,Z 332.324,A -85,B 0,C 180,E1 -15357.428,E2 -15357.428} C_VEL
LIN {X 0,Y 322.274,Z 335.513,A -85,B 0,C 180,E1 -15357.671,E2 -15357.671} C_VEL
LIN {X 0,Y 328.65,Z 349.657,A -85,B 0,C 180,E1 -15358.883,E2 -15358.883} C_VEL
LIN {X 0,Y 333.73,Z 363.389,A -85,B 0,C 180,E1 -15360.142,E2 -15360.142} C_VEL
LIN {X 0,Y 337.421,Z 375.841,A -85,B 0,C 180,E1 -15361.376,E2 -15361.376} C_VEL
LIN {X 0,Y 337.396,Z 379.355,A -85,B 0,C 180,E1 -15361.65,E2 -15361.65} C_VEL
LIN {X 0,Y 335.809,Z 392.992,A -85,B 0,C 180,E1 -15362.754,E2 -15362.754} C_VEL
LIN {X 0,Y 333.819,Z 406.393,A -85,B 0,C 180,E1 -15364.096,E2 -15364.096} C_VEL
LIN {X 0,Y 331.607,Z 418.752,A -85,B 0,C 180,E1 -15365.607,E2 -15365.607} C_VEL
LIN {X 0,Y 329.741,Z 428.901,A -85,B 0,C 180,E1 -15367.109,E2 -15367.109} C_VEL
LIN {X 0,Y 327.639,Z 439.356,A -85,B 0,C 180,E1 -15368.943,E2 -15368.943} C_VEL
LIN {X 0,Y 325.434,Z 449.523,A -85,B 0,C 180,E1 -15371.099,E2 -15371.099} C_VEL
LIN {X 0,Y 323.572,Z 457.927,A -85,B 0,C 180,E1 -15373.264,E2 -15373.264} C_VEL
LIN {X 0,Y 322.088,Z 464.957,A -85,B 0,C 180,E1 -15375.467,E2 -15375.467} C_VEL
LIN {X 0,Y 320.769,Z 471.416,A -85,B 0,C 180,E1 -15377.986,E2 -15377.986} C_VEL
LIN {X 0,Y 319.753,Z 476.463,A -85,B 0,C 180,E1 -15380.511,E2 -15380.511} C_VEL
LIN {X 0,Y 319.216,Z 479.359,A -85,B 0,C 180,E1 -15382.409,E2 -15382.409} C_VEL
LIN {X 0,Y 318.83,Z 482.195,A -85,B 0,C 180,E1 -15384.941,E2 -15384.941} C_VEL
LIN {X 0,Y 318.575,Z 483.896,A -85,B 0,C 180,E1 -15387.471,E2 -15387.471} C_VEL
LIN {X 0,Y 318.422,Z 484.492,A -85,B 0,C 180,E1 -15390,E2 -15390} C_VEL
LIN {X 0,Y 318.57,Z 483.933,A -85,B 0,C 180,E1 -15392.529,E2 -15392.529} C_VEL
LIN {X 0,Y 318.828,Z 482.281,A -85,B 0,C 180,E1 -15395.058,E2 -15395.058} C_VEL
LIN {X 0,Y 319.215,Z 479.502,A -85,B 0,C 180,E1 -15397.591,E2 -15397.591} C_VEL
LIN {X 0,Y 319.941,Z 475.51,A -85,B 0,C 180,E1 -15400.121,E2 -15400.121} C_VEL
LIN {X 0,Y 321.032,Z 470.192,A -85,B 0,C 180,E1 -15402.645,E2 -15402.645} C_VEL
LIN {X 0,Y 322.424,Z 463.406,A -85,B 0,C 180,E1 -15405.163,E2 -15405.163} C_VEL
LIN {X 0,Y 324.027,Z 456.015,A -85,B 0,C 180,E1 -15407.38,E2 -15407.38} C_VEL
LIN {X 0,Y 325.978,Z 447.32,A -85,B 0,C 180,E1 -15409.522,E2 -15409.522} C_VEL
LIN {X 0,Y 328.267,Z 436.657,A -85,B 0,C 180,E1 -15411.673,E2 -15411.673} C_VEL
LIN {X 0,Y 330.255,Z 425.739,A -85,B 0,C 180,E1 -15413.511,E2 -15413.511} C_VEL
LIN {X 0,Y 332.611,Z 413.635,A -85,B 0,C 180,E1 -15415.165,E2 -15415.165} C_VEL
LIN {X 0,Y 334.763,Z 400.295,A -85,B 0,C 180,E1 -15416.663,E2 -15416.663} C_VEL
LIN {X 0,Y 336.525,Z 387.555,A -85,B 0,C 180,E1 -15417.828,E2 -15417.828} C_VEL
LIN {X 0,Y 337.652,Z 377.239,A -85,B 0,C 180,E1 -15418.602,E2 -15418.602} C_VEL
LIN {X 0,Y 334.169,Z 364.632,A -85,B 0,C 180,E1 -15419.851,E2 -15419.851} C_VEL
LIN {X 0,Y 329.179,Z 350.72,A -85,B 0,C 180,E1 -15421.129,E2 -15421.129} C_VEL
LIN {X 0,Y 322.489,Z 335.84,A -85,B 0,C 180,E1 -15422.411,E2 -15422.411} C_VEL
LIN {X 0,Y 321.04,Z 332.815,A -85,B 0,C 180,E1 -15422.658,E2 -15422.658} C_VEL
LIN {X 0,Y 320.922,Z 332.262,A -85,B 0,C 180,E1 -15422.735,E2 -15422.735} C_VEL
LIN {X 0,Y 320.917,Z 327.355,A -85,B 0,C 180,E1 -15426.249,E2 -15426.249} C_VEL
LIN {X 0,Y 320.995,Z 323.221,A -85,B 0,C 180,E1 -15429.415,E2 -15429.415} C_VEL
LIN {X 0,Y 320.837,Z 319.043,A -85,B 0,C 180,E1 -15432.77,E2 -15432.77} C_VEL
LIN {X 0,Y 320.394,Z 315.91,A -85,B 0,C 180,E1 -15435.417,E2 -15435.417} C_VEL
LIN {X 0,Y 319.566,Z 311.39,A -85,B 0,C 180,E1 -15439.344,E2 -15439.344} C_VEL
LIN {X 0,Y 319.573,Z 311.304,A -85,B 0,C 180,E1 -15442.154,E2 -15442.154} C_VEL
LIN {X 0,Y 318.919,Z 311.387,A -85,B 0,C 180,E1 -15443.207,E2 -15443.207} C_VEL
LIN {X 0,Y 316.064,Z 311.743,A -85,B 0,C 180,E1 -15444.919,E2 -15444.919} C_VEL
LIN {X 0,Y 313.628,Z 312.041,A -85,B 0,C 180,E1 -15446.308,E2 -15446.308} C_VEL
LIN {X 0,Y 312.572,Z 312.17,A -85,B 0,C 180,E1 -15447.383,E2 -15447.383} C_VEL
LIN {X 0,Y 312.482,Z 312.179,A -85,B 0,C 180,E1 -15447.747,E2 -15447.747} C_VEL
LIN {X 0,Y 312.526,Z 312.182,A -85,B 0,C 180,E1 -15451.82,E2 -15451.82} C_VEL
LIN {X 0,Y 312.546,Z 312.168,A -85,B 0,C 180,E1 -15454.707,E2 -15454.707} C_VEL
LIN {X 0,Y 312.534,Z 312.165,A -85,B 0,C 180,E1 -15458.912,E2 -15458.912} C_VEL
LIN {X 0,Y 312.588,Z 312.166,A -85,B 0,C 180,E1 -15461.653,E2 -15461.653} C_VEL
LIN {X 0,Y 312.685,Z 312.162,A -85,B 0,C 180,E1 -15465.686,E2 -15465.686} C_VEL
LIN {X 0,Y 312.685,Z 312.149,A -85,B 0,C 180,E1 -15469.641,E2 -15469.641} C_VEL
LIN {X 0,Y 312.796,Z 312.141,A -85,B 0,C 180,E1 -15472.252,E2 -15472.252} C_VEL
LIN {X 0,Y 312.7,Z 312.141,A -85,B 0,C 180,E1 -15474.842,E2 -15474.842} C_VEL
LIN {X 0,Y 312.991,Z 312.105,A -85,B 0,C 180,E1 -15478.713,E2 -15478.713} C_VEL
LIN {X 0,Y 312.987,Z 312.116,A -85,B 0,C 180,E1 -15481.287,E2 -15481.287} C_VEL
LIN {X 0,Y 312.698,Z 312.137,A -85,B 0,C 180,E1 -15485.158,E2 -15485.158} C_VEL
LIN {X 0,Y 312.828,Z 312.142,A -85,B 0,C 180,E1 -15487.747,E2 -15487.747} C_VEL
LIN {X 0,Y 312.664,Z 312.143,A -85,B 0,C 180,E1 -15491.671,E2 -15491.671} C_VEL
LIN {X 0,Y 312.7,Z 312.151,A -85,B 0,C 180,E1 -15494.888,E2 -15494.888} C_VEL
LIN {X 0,Y 312.629,Z 312.169,A -85,B 0,C 180,E1 -15499.236,E2 -15499.236} C_VEL
LIN {X 0,Y 312.521,Z 312.17,A -85,B 0,C 180,E1 -15502.779,E2 -15502.779} C_VEL
LIN {X 0,Y 312.529,Z 312.166,A -85,B 0,C 180,E1 -15505.908,E2 -15505.908} C_VEL
LIN {X 0,Y 312.495,Z 312.185,A -85,B 0,C 180,E1 -15509.655,E2 -15509.655} C_VEL
LIN {X 0,Y 312.518,Z 312.182,A -85,B 0,C 180,E1 -15513.689,E2 -15513.689} C_VEL
LIN {X 0,Y 312.556,Z 312.346,A -85,B 0,C 180,E1 -15514.986,E2 -15514.986} C_VEL
LIN {X 0,Y 314.336,Z 320.138,A -85,B 0,C 180,E1 -15518.758,E2 -15518.758} C_VEL
LIN {X 0,Y 316.155,Z 328.105,A -85,B 0,C 180,E1 -15522.365,E2 -15522.365} C_VEL
LIN {X 0,Y 318.356,Z 337.435,A -85,B 0,C 180,E1 -15526.301,E2 -15526.301} C_VEL
LIN {X 0,Y 320.621,Z 347.052,A -85,B 0,C 180,E1 -15530.103,E2 -15530.103} C_VEL
LIN {X 0,Y 321.693,Z 351.671,A -85,B 0,C 180,E1 -15531.858,E2 -15531.858} C_VEL
LIN {X 0,Y 321.218,Z 355.028,A -85,B 0,C 180,E1 -15533.01,E2 -15533.01} C_VEL
LIN {X 0,Y 319.023,Z 364.52,A -85,B 0,C 180,E1 -15536.108,E2 -15536.108} C_VEL
LIN {X 0,Y 318.933,Z 371.273,A -85,B 0,C 180,E1 -15537.184,E2 -15537.184} C_VEL
LIN {X 0,Y 322.474,Z 387.735,A -85,B 0,C 180,E1 -15538.022,E2 -15538.022} C_VEL
LIN {X 0,Y 324.944,Z 403.58,A -85,B 0,C 180,E1 -15538.911,E2 -15538.911} C_VEL
LIN {X 0,Y 326.399,Z 418.688,A -85,B 0,C 180,E1 -15539.933,E2 -15539.933} C_VEL
LIN {X 0,Y 327.173,Z 433.001,A -85,B 0,C 180,E1 -15541.098,E2 -15541.098} C_VEL
LIN {X 0,Y 326.966,Z 438.883,A -85,B 0,C 180,E1 -15541.604,E2 -15541.604} C_VEL
LIN {X 0,Y 324.903,Z 451.841,A -85,B 0,C 180,E1 -15542.774,E2 -15542.774} C_VEL
LIN {X 0,Y 322.316,Z 465.638,A -85,B 0,C 180,E1 -15544.319,E2 -15544.319} C_VEL
LIN {X 0,Y 319.868,Z 477.925,A -85,B 0,C 180,E1 -15546.017,E2 -15546.017} C_VEL
LIN {X 0,Y 317.673,Z 489.166,A -85,B 0,C 180,E1 -15547.908,E2 -15547.908} C_VEL
LIN {X 0,Y 315.783,Z 498.65,A -85,B 0,C 180,E1 -15549.821,E2 -15549.821} C_VEL
LIN {X 0,Y 313.989,Z 507.976,A -85,B 0,C 180,E1 -15552.076,E2 -15552.076} C_VEL
LIN {X 0,Y 312.7,Z 515.745,A -85,B 0,C 180,E1 -15554.354,E2 -15554.354} C_VEL
LIN {X 0,Y 311.675,Z 523.02,A -85,B 0,C 180,E1 -15556.969,E2 -15556.969} C_VEL
LIN {X 0,Y 311.182,Z 528.768,A -85,B 0,C 180,E1 -15559.591,E2 -15559.591} C_VEL
LIN {X 0,Y 311.078,Z 533.128,A -85,B 0,C 180,E1 -15562.21,E2 -15562.21} C_VEL
LIN {X 0,Y 311.221,Z 534.829,A -85,B 0,C 180,E1 -15563.517,E2 -15563.517} C_VEL
LIN {X 0,Y 311.221,Z 537.266,A -85,B 0,C 180,E1 -15566.116,E2 -15566.116} C_VEL
LIN {X 0,Y 311.391,Z 538.043,A -85,B 0,C 180,E1 -15567.413,E2 -15567.413} C_VEL
LIN {X 0,Y 311.493,Z 538.673,A -85,B 0,C 180,E1 -15570,E2 -15570} C_VEL
LIN {X 0,Y 311.411,Z 538.041,A -85,B 0,C 180,E1 -15572.587,E2 -15572.587} C_VEL
LIN {X 0,Y 311.239,Z 536.194,A -85,B 0,C 180,E1 -15575.182,E2 -15575.182} C_VEL
LIN {X 0,Y 311.138,Z 533.112,A -85,B 0,C 180,E1 -15577.789,E2 -15577.789} C_VEL
LIN {X 0,Y 311.205,Z 528.734,A -85,B 0,C 180,E1 -15580.409,E2 -15580.409} C_VEL
LIN {X 0,Y 311.708,Z 522.98,A -85,B 0,C 180,E1 -15583.031,E2 -15583.031} C_VEL
LIN {X 0,Y 312.707,Z 515.697,A -85,B 0,C 180,E1 -15585.647,E2 -15585.647} C_VEL
LIN {X 0,Y 313.975,Z 507.911,A -85,B 0,C 180,E1 -15587.926,E2 -15587.926} C_VEL
LIN {X 0,Y 315.848,Z 498.572,A -85,B 0,C 180,E1 -15590.176,E2 -15590.176} C_VEL
LIN {X 0,Y 317.688,Z 489.074,A -85,B 0,C 180,E1 -15592.091,E2 -15592.091} C_VEL
LIN {X 0,Y 320.126,Z 476.779,A -85,B 0,C 180,E1 -15594.135,E2 -15594.135} C_VEL
LIN {X 0,Y 322.593,Z 464.481,A -85,B 0,C 180,E1 -15595.831,E2 -15595.831} C_VEL
LIN {X 0,Y 326.231,Z 451.241,A -85,B 0,C 180,E1 -15597.742,E2 -15597.742} C_VEL
LIN {X 0,Y 329.43,Z 439.249,A -85,B 0,C 180,E1 -15599.193,E2 -15599.193} C_VEL
LIN {X 0,Y 331.468,Z 424.287,A -85,B 0,C 180,E1 -15600.968,E2 -15600.968} C_VEL
LIN {X 0,Y 332.203,Z 412.642,A -85,B 0,C 180,E1 -15602.301,E2 -15602.301} C_VEL
LIN {X 0,Y 331.632,Z 398.526,A -85,B 0,C 180,E1 -15604.061,E2 -15604.061} C_VEL
LIN {X 0,Y 330.263,Z 386.072,A -85,B 0,C 180,E1 -15605.77,E2 -15605.77} C_VEL
LIN {X 0,Y 328.431,Z 375.101,A -85,B 0,C 180,E1 -15607.476,E2 -15607.476} C_VEL
LIN {X 0,Y 327.68,Z 370.131,A -85,B 0,C 180,E1 -15608.293,E2 -15608.293} C_VEL
LIN {X 0,Y 326.263,Z 366.274,A -85,B 0,C 180,E1 -15609.262,E2 -15609.262} C_VEL
LIN {X 0,Y 324.917,Z 362.492,A -85,B 0,C 180,E1 -15610.36,E2 -15610.36} C_VEL
LIN {X 0,Y 323.407,Z 357.48,A -85,B 0,C 180,E1 -15614.059,E2 -15614.059} C_VEL
LIN {X 0,Y 322.257,Z 354.001,A -85,B 0,C 180,E1 -15617.463,E2 -15617.463} C_VEL
LIN {X 0,Y 321.299,Z 351.682,A -85,B 0,C 180,E1 -15620.629,E2 -15620.629} C_VEL
LIN {X 0,Y 320.853,Z 350.887,A -85,B 0,C 180,E1 -15622.434,E2 -15622.434} C_VEL
LIN {X 0,Y 321.818,Z 352.595,A -85,B 0,C 180,E1 -15623.904,E2 -15623.904} C_VEL
LIN {X 0,Y 323.766,Z 354.285,A -85,B 0,C 180,E1 -15625.641,E2 -15625.641} C_VEL
LIN {X 0,Y 324.663,Z 355.849,A -85,B 0,C 180,E1 -15626.478,E2 -15626.478} C_VEL
LIN {X 0,Y 325.998,Z 357.09,A -85,B 0,C 180,E1 -15627.387,E2 -15627.387} C_VEL
LIN {X 0,Y 329.692,Z 363.058,A -85,B 0,C 180,E1 -15629.964,E2 -15629.964} C_VEL
LIN {X 0,Y 333.297,Z 370.085,A -85,B 0,C 180,E1 -15632.329,E2 -15632.329} C_VEL
LIN {X 0,Y 335.901,Z 376.448,A -85,B 0,C 180,E1 -15634.117,E2 -15634.117} C_VEL
LIN {X 0,Y 337.452,Z 382.323,A -85,B 0,C 180,E1 -15635.514,E2 -15635.514} C_VEL
LIN {X 0,Y 334.095,Z 394.046,A -85,B 0,C 180,E1 -15637.098,E2 -15637.098} C_VEL
LIN {X 0,Y 330.891,Z 404.44,A -85,B 0,C 180,E1 -15638.834,E2 -15638.834} C_VEL
LIN {X 0,Y 327.533,Z 414.319,A -85,B 0,C 180,E1 -15640.85,E2 -15640.85} C_VEL
LIN {X 0,Y 324.833,Z 421.626,A -85,B 0,C 180,E1 -15642.693,E2 -15642.693} C_VEL
LIN {X 0,Y 322.164,Z 428.429,A -85,B 0,C 180,E1 -15644.824,E2 -15644.824} C_VEL
LIN {X 0,Y 320.111,Z 433.145,A -85,B 0,C 180,E1 -15646.672,E2 -15646.672} C_VEL
LIN {X 0,Y 317.881,Z 437.919,A -85,B 0,C 180,E1 -15649.168,E2 -15649.168} C_VEL
LIN {X 0,Y 316.439,Z 440.452,A -85,B 0,C 180,E1 -15651.056,E2 -15651.056} C_VEL
LIN {X 0,Y 315.663,Z 441.65,A -85,B 0,C 180,E1 -15652.323,E2 -15652.323} C_VEL
LIN {X 0,Y 314.578,Z 442.84,A -85,B 0,C 180,E1 -15654.873,E2 -15654.873} C_VEL
LIN {X 0,Y 313.58,Z 442.626,A -85,B 0,C 180,E1 -15657.431,E2 -15657.431} C_VEL
LIN {X 0,Y 313.336,Z 441.924,A -85,B 0,C 180,E1 -15658.715,E2 -15658.715} C_VEL
LIN {X 0,Y 312.904,Z 440.841,A -85,B 0,C 180,E1 -15660,E2 -15660} C_VEL
LIN {X 0,Y 312.872,Z 439.324,A -85,B 0,C 180,E1 -15661.287,E2 -15661.287} C_VEL
LIN {X 0,Y 312.626,Z 436.346,A -85,B 0,C 180,E1 -15663.222,E2 -15663.222} C_VEL
LIN {X 0,Y 312.764,Z 432.371,A -85,B 0,C 180,E1 -15665.157,E2 -15665.157} C_VEL
LIN {X 0,Y 313.193,Z 427.351,A -85,B 0,C 180,E1 -15667.09,E2 -15667.09} C_VEL
LIN {X 0,Y 313.666,Z 420.032,A -85,B 0,C 180,E1 -15669.352,E2 -15669.352} C_VEL
LIN {X 0,Y 314.285,Z 412.361,A -85,B 0,C 180,E1 -15671.284,E2 -15671.284} C_VEL
LIN {X 0,Y 315.048,Z 403.11,A -85,B 0,C 180,E1 -15673.218,E2 -15673.218} C_VEL
LIN {X 0,Y 316.04,Z 391.778,A -85,B 0,C 180,E1 -15675.147,E2 -15675.147} C_VEL
LIN {X 0,Y 317.124,Z 380.386,A -85,B 0,C 180,E1 -15676.745,E2 -15676.745} C_VEL
LIN {X 0,Y 318.141,Z 367.604,A -85,B 0,C 180,E1 -15678.211,E2 -15678.211} C_VEL
LIN {X 0,Y 319.144,Z 354.773,A -85,B 0,C 180,E1 -15679.406,E2 -15679.406} C_VEL
LIN {X 0,Y 319.059,Z 351.911,A -85,B 0,C 180,E1 -15679.648,E2 -15679.648} C_VEL
LIN {X 0,Y 315.657,Z 337.399,A -85,B 0,C 180,E1 -15680.869,E2 -15680.869} C_VEL
LIN {X 0,Y 312.025,Z 322.685,A -85,B 0,C 180,E1 -15681.861,E2 -15681.861} C_VEL
LIN {X 0,Y 311.991,Z 318.711,A -85,B 0,C 180,E1 -15685.703,E2 -15685.703} C_VEL
LIN {X 0,Y 312.046,Z 315.833,A -85,B 0,C 180,E1 -15688.553,E2 -15688.553} C_VEL
LIN {X 0,Y 312.074,Z 313.23,A -85,B 0,C 180,E1 -15691.196,E2 -15691.196} C_VEL
LIN {X 0,Y 312.092,Z 312.237,A -85,B 0,C 180,E1 -15692.715,E2 -15692.715} C_VEL
LIN {X 0,Y 312.44,Z 312.192,A -85,B 0,C 180,E1 -15695.925,E2 -15695.925} C_VEL
LIN {X 0,Y 312.541,Z 312.236,A -85,B 0,C 180,E1 -15699.866,E2 -15699.866} C_VEL
LIN {X 0,Y 313.061,Z 315,A -85,B 0,C 180,E1 -15702.336,E2 -15702.336} C_VEL
LIN {X 0,Y 313.785,Z 319.186,A -85,B 0,C 180,E1 -15706.026,E2 -15706.026} C_VEL
LIN {X 0,Y 314.088,Z 322.424,A -85,B 0,C 180,E1 -15708.694,E2 -15708.694} C_VEL
LIN {X 0,Y 314.087,Z 326.023,A -85,B 0,C 180,E1 -15711.551,E2 -15711.551} C_VEL
LIN {X 0,Y 314.044,Z 330.909,A -85,B 0,C 180,E1 -15715.204,E2 -15715.204} C_VEL
LIN {X 0,Y 314.019,Z 332.935,A -85,B 0,C 180,E1 -15716.624,E2 -15716.624} C_VEL
LIN {X 0,Y 315.393,Z 336.165,A -85,B 0,C 180,E1 -15716.878,E2 -15716.878} C_VEL
LIN {X 0,Y 321.936,Z 350.33,A -85,B 0,C 180,E1 -15718.161,E2 -15718.161} C_VEL
LIN {X 0,Y 327.055,Z 364.118,A -85,B 0,C 180,E1 -15719.475,E2 -15719.475} C_VEL
LIN {X 0,Y 330.772,Z 376.472,A -85,B 0,C 180,E1 -15720.745,E2 -15720.745} C_VEL
LIN {X 0,Y 331.268,Z 378.429,A -85,B 0,C 180,E1 -15720.955,E2 -15720.955} C_VEL
LIN {X 0,Y 329.778,Z 391.877,A -85,B 0,C 180,E1 -15722.04,E2 -15722.04} C_VEL
LIN {X 0,Y 327.702,Z 405.61,A -85,B 0,C 180,E1 -15723.404,E2 -15723.404} C_VEL
LIN {X 0,Y 325.337,Z 418.29,A -85,B 0,C 180,E1 -15724.946,E2 -15724.946} C_VEL
LIN {X 0,Y 323.241,Z 429.504,A -85,B 0,C 180,E1 -15726.622,E2 -15726.622} C_VEL
LIN {X 0,Y 321.057,Z 439.96,A -85,B 0,C 180,E1 -15728.49,E2 -15728.49} C_VEL
LIN {X 0,Y 318.737,Z 450.131,A -85,B 0,C 180,E1 -15730.686,E2 -15730.686} C_VEL
LIN {X 0,Y 316.759,Z 458.643,A -85,B 0,C 180,E1 -15732.926,E2 -15732.926} C_VEL
LIN {X 0,Y 315.237,Z 465.566,A -85,B 0,C 180,E1 -15735.144,E2 -15735.144} C_VEL
LIN {X 0,Y 313.838,Z 472.025,A -85,B 0,C 180,E1 -15737.717,E2 -15737.717} C_VEL
LIN {X 0,Y 312.768,Z 477.073,A -85,B 0,C 180,E1 -15740.297,E2 -15740.297} C_VEL
LIN {X 0,Y 312.222,Z 479.966,A -85,B 0,C 180,E1 -15742.238,E2 -15742.238} C_VEL
LIN {X 0,Y 311.781,Z 482.804,A -85,B 0,C 180,E1 -15744.827,E2 -15744.827} C_VEL
LIN {X 0,Y 311.518,Z 484.504,A -85,B 0,C 180,E1 -15747.414,E2 -15747.414} C_VEL
LIN {X 0,Y 311.354,Z 485.1,A -85,B 0,C 180,E1 -15750,E2 -15750} C_VEL
LIN {X 0,Y 311.512,Z 484.54,A -85,B 0,C 180,E1 -15752.586,E2 -15752.586} C_VEL
LIN {X 0,Y 311.762,Z 482.89,A -85,B 0,C 180,E1 -15755.173,E2 -15755.173} C_VEL
LIN {X 0,Y 312.312,Z 479.721,A -85,B 0,C 180,E1 -15758.052,E2 -15758.052} C_VEL
LIN {X 0,Y 312.981,Z 476.116,A -85,B 0,C 180,E1 -15760.349,E2 -15760.349} C_VEL
LIN {X 0,Y 314.124,Z 470.798,A -85,B 0,C 180,E1 -15762.928,E2 -15762.928} C_VEL
LIN {X 0,Y 315.59,Z 464.012,A -85,B 0,C 180,E1 -15765.499,E2 -15765.499} C_VEL
LIN {X 0,Y 317.21,Z 456.879,A -85,B 0,C 180,E1 -15767.694,E2 -15767.694} C_VEL
LIN {X 0,Y 319.312,Z 447.922,A -85,B 0,C 180,E1 -15769.947,E2 -15769.947} C_VEL
LIN {X 0,Y 321.685,Z 437.258,A -85,B 0,C 180,E1 -15772.14,E2 -15772.14} C_VEL
LIN {X 0,Y 323.77,Z 426.396,A -85,B 0,C 180,E1 -15774.001,E2 -15774.001} C_VEL
LIN {X 0,Y 326.221,Z 414.227,A -85,B 0,C 180,E1 -15775.694,E2 -15775.694} C_VEL
LIN {X 0,Y 328.477,Z 400.879,A -85,B 0,C 180,E1 -15777.215,E2 -15777.215} C_VEL
LIN {X 0,Y 330.402,Z 387.346,A -85,B 0,C 180,E1 -15778.461,E2 -15778.461} C_VEL
LIN {X 0,Y 331.372,Z 378.855,A -85,B 0,C 180,E1 -15779.112,E2 -15779.112} C_VEL
LIN {X 0,Y 327.482,Z 365.265,A -85,B 0,C 180,E1 -15780.523,E2 -15780.523} C_VEL
LIN {X 0,Y 322.658,Z 351.916,A -85,B 0,C 180,E1 -15781.804,E2 -15781.804} C_VEL
LIN {X 0,Y 316.458,Z 338.379,A -85,B 0,C 180,E1 -15783.049,E2 -15783.049} C_VEL
LIN {X 0,Y 314.154,Z 333.494,A -85,B 0,C 180,E1 -15783.463,E2 -15783.463} C_VEL
LIN {X 0,Y 314.014,Z 332.907,A -85,B 0,C 180,E1 -15783.52,E2 -15783.52} C_VEL
LIN {X 0,Y 314.025,Z 329.011,A -85,B 0,C 180,E1 -15786.323,E2 -15786.323} C_VEL
LIN {X 0,Y 314.108,Z 324.742,A -85,B 0,C 180,E1 -15789.618,E2 -15789.618} C_VEL
LIN {X 0,Y 313.994,Z 321.264,A -85,B 0,C 180,E1 -15792.385,E2 -15792.385} C_VEL
LIN {X 0,Y 313.745,Z 319.075,A -85,B 0,C 180,E1 -15794.208,E2 -15794.208} C_VEL
LIN {X 0,Y 313.042,Z 315.003,A -85,B 0,C 180,E1 -15797.806,E2 -15797.806} C_VEL
LIN {X 0,Y 312.514,Z 312.178,A -85,B 0,C 180,E1 -15800.408,E2 -15800.408} C_VEL
LIN {X 0,Y 312.532,Z 312.176,A -85,B 0,C 180,E1 -15804.22,E2 -15804.22} C_VEL
LIN {X 0,Y 312.482,Z 312.179,A -85,B 0,C 180,E1 -15807.747,E2 -15807.747} C_VEL
LIN {X 0,Y 311.798,Z 312.268,A -85,B 0,C 180,E1 -15808.823,E2 -15808.823} C_VEL
LIN {X 0,Y 308.931,Z 312.623,A -85,B 0,C 180,E1 -15810.574,E2 -15810.574} C_VEL
LIN {X 0,Y 306.526,Z 312.93,A -85,B 0,C 180,E1 -15811.995,E2 -15811.995} C_VEL
LIN {X 0,Y 305.519,Z 313.044,A -85,B 0,C 180,E1 -15813.094,E2 -15813.094} C_VEL
LIN {X 0,Y 305.45,Z 313.049,A -85,B 0,C 180,E1 -15813.467,E2 -15813.467} C_VEL
LIN {X 0,Y 305.491,Z 313.05,A -85,B 0,C 180,E1 -15816.977,E2 -15816.977} C_VEL
LIN {X 0,Y 305.548,Z 313.049,A -85,B 0,C 180,E1 -15821.215,E2 -15821.215} C_VEL
LIN {X 0,Y 305.626,Z 313.04,A -85,B 0,C 180,E1 -15825.348,E2 -15825.348} C_VEL
LIN {X 0,Y 305.624,Z 313.025,A -85,B 0,C 180,E1 -15829.399,E2 -15829.399} C_VEL
LIN {X 0,Y 305.746,Z 313.02,A -85,B 0,C 180,E1 -15832.072,E2 -15832.072} C_VEL
LIN {X 0,Y 305.668,Z 313.015,A -85,B 0,C 180,E1 -15834.723,E2 -15834.723} C_VEL
LIN {X 0,Y 305.957,Z 312.98,A -85,B 0,C 180,E1 -15838.684,E2 -15838.684} C_VEL
LIN {X 0,Y 305.953,Z 312.991,A -85,B 0,C 180,E1 -15841.316,E2 -15841.316} C_VEL
LIN {X 0,Y 305.804,Z 313.004,A -85,B 0,C 180,E1 -15846.598,E2 -15846.598} C_VEL
LIN {X 0,Y 305.694,Z 313.025,A -85,B 0,C 180,E1 -15849.261,E2 -15849.261} C_VEL
LIN {X 0,Y 305.589,Z 313.044,A -85,B 0,C 180,E1 -15853.296,E2 -15853.296} C_VEL
LIN {X 0,Y 305.593,Z 313.024,A -85,B 0,C 180,E1 -15856.02,E2 -15856.02} C_VEL
LIN {X 0,Y 305.575,Z 313.047,A -85,B 0,C 180,E1 -15859.444,E2 -15859.444} C_VEL
LIN {X 0,Y 305.485,Z 313.049,A -85,B 0,C 180,E1 -15863.039,E2 -15863.039} C_VEL
LIN {X 0,Y 305.469,Z 313.043,A -85,B 0,C 180,E1 -15866.197,E2 -15866.197} C_VEL
LIN {X 0,Y 305.448,Z 313.063,A -85,B 0,C 180,E1 -15869.034,E2 -15869.034} C_VEL
LIN {X 0,Y 305.435,Z 313.064,A -85,B 0,C 180,E1 -15871.953,E2 -15871.953} C_VEL
LIN {X 0,Y 305.489,Z 313.09,A -85,B 0,C 180,E1 -15874.246,E2 -15874.246} C_VEL
LIN {X 0,Y 307.226,Z 320.865,A -85,B 0,C 180,E1 -15878.144,E2 -15878.144} C_VEL
LIN {X 0,Y 309.183,Z 329.421,A -85,B 0,C 180,E1 -15882.109,E2 -15882.109} C_VEL
LIN {X 0,Y 311.427,Z 338.932,A -85,B 0,C 180,E1 -15886.232,E2 -15886.232} C_VEL
LIN {X 0,Y 313.874,Z 349.391,A -85,B 0,C 180,E1 -15890.46,E2 -15890.46} C_VEL
LIN {X 0,Y 314.491,Z 351.986,A -85,B 0,C 180,E1 -15891.458,E2 -15891.458} C_VEL
LIN {X 0,Y 314.655,Z 353.979,A -85,B 0,C 180,E1 -15892.2,E2 -15892.2} C_VEL
LIN {X 0,Y 312.65,Z 362.142,A -85,B 0,C 180,E1 -15894.977,E2 -15894.977} C_VEL
LIN {X 0,Y 312.443,Z 370.629,A -85,B 0,C 180,E1 -15896.41,E2 -15896.41} C_VEL
LIN {X 0,Y 316.074,Z 387.442,A -85,B 0,C 180,E1 -15897.302,E2 -15897.302} C_VEL
LIN {X 0,Y 318.591,Z 403.454,A -85,B 0,C 180,E1 -15898.243,E2 -15898.243} C_VEL
LIN {X 0,Y 320.045,Z 419.08,A -85,B 0,C 180,E1 -15899.341,E2 -15899.341} C_VEL
LIN {X 0,Y 320.74,Z 433.404,A -85,B 0,C 180,E1 -15900.551,E2 -15900.551} C_VEL
LIN {X 0,Y 320.243,Z 441.178,A -85,B 0,C 180,E1 -15901.244,E2 -15901.244} C_VEL
LIN {X 0,Y 317.966,Z 454.411,A -85,B 0,C 180,E1 -15902.523,E2 -15902.523} C_VEL
LIN {X 0,Y 315.413,Z 467.401,A -85,B 0,C 180,E1 -15904.07,E2 -15904.07} C_VEL
LIN {X 0,Y 312.895,Z 479.289,A -85,B 0,C 180,E1 -15905.801,E2 -15905.801} C_VEL
LIN {X 0,Y 310.672,Z 490.119,A -85,B 0,C 180,E1 -15907.716,E2 -15907.716} C_VEL
LIN {X 0,Y 308.725,Z 499.472,A -85,B 0,C 180,E1 -15909.687,E2 -15909.687} C_VEL
LIN {X 0,Y 306.905,Z 508.57,A -85,B 0,C 180,E1 -15911.993,E2 -15911.993} C_VEL
LIN {X 0,Y 305.448,Z 517.112,A -85,B 0,C 180,E1 -15914.658,E2 -15914.658} C_VEL
LIN {X 0,Y 304.515,Z 523.989,A -85,B 0,C 180,E1 -15917.335,E2 -15917.335} C_VEL
LIN {X 0,Y 304.064,Z 529.391,A -85,B 0,C 180,E1 -15920.018,E2 -15920.018} C_VEL
LIN {X 0,Y 303.997,Z 532.514,A -85,B 0,C 180,E1 -15922.027,E2 -15922.027} C_VEL
LIN {X 0,Y 304.135,Z 534.413,A -85,B 0,C 180,E1 -15923.538,E2 -15923.538} C_VEL
LIN {X 0,Y 304.136,Z 536.656,A -85,B 0,C 180,E1 -15926.025,E2 -15926.025} C_VEL
LIN {X 0,Y 304.324,Z 537.434,A -85,B 0,C 180,E1 -15927.353,E2 -15927.353} C_VEL
LIN {X 0,Y 304.419,Z 538.065,A -85,B 0,C 180,E1 -15930,E2 -15930} C_VEL
LIN {X 0,Y 304.343,Z 537.432,A -85,B 0,C 180,E1 -15932.647,E2 -15932.647} C_VEL
LIN {X 0,Y 304.173,Z 535.584,A -85,B 0,C 180,E1 -15935.303,E2 -15935.303} C_VEL
LIN {X 0,Y 304.044,Z 532.496,A -85,B 0,C 180,E1 -15937.972,E2 -15937.972} C_VEL
LIN {X 0,Y 304.139,Z 528.116,A -85,B 0,C 180,E1 -15940.653,E2 -15940.653} C_VEL
LIN {X 0,Y 304.701,Z 522.362,A -85,B 0,C 180,E1 -15943.336,E2 -15943.336} C_VEL
LIN {X 0,Y 305.784,Z 515.079,A -85,B 0,C 180,E1 -15946.01,E2 -15946.01} C_VEL
LIN {X 0,Y 307.129,Z 507.293,A -85,B 0,C 180,E1 -15948.339,E2 -15948.339} C_VEL
LIN {X 0,Y 309.118,Z 497.957,A -85,B 0,C 180,E1 -15950.635,E2 -15950.635} C_VEL
LIN {X 0,Y 311.032,Z 488.459,A -85,B 0,C 180,E1 -15952.59,E2 -15952.59} C_VEL
LIN {X 0,Y 313.58,Z 476.167,A -85,B 0,C 180,E1 -15954.673,E2 -15954.673} C_VEL
LIN {X 0,Y 315.172,Z 468.683,A -85,B 0,C 180,E1 -15955.775,E2 -15955.775} C_VEL
LIN {X 0,Y 319.069,Z 455.749,A -85,B 0,C 180,E1 -15957.845,E2 -15957.845} C_VEL
LIN {X 0,Y 323.051,Z 442.226,A -85,B 0,C 180,E1 -15959.629,E2 -15959.629} C_VEL
LIN {X 0,Y 325.597,Z 427.691,A -85,B 0,C 180,E1 -15961.445,E2 -15961.445} C_VEL
LIN {X 0,Y 326.826,Z 414.943,A -85,B 0,C 180,E1 -15963.003,E2 -15963.003} C_VEL
LIN {X 0,Y 326.683,Z 401.243,A -85,B 0,C 180,E1 -15964.816,E2 -15964.816} C_VEL
LIN {X 0,Y 325.868,Z 390.185,A -85,B 0,C 180,E1 -15966.424,E2 -15966.424} C_VEL
LIN {X 0,Y 324.59,Z 379.707,A -85,B 0,C 180,E1 -15968.146,E2 -15968.146} C_VEL
LIN {X 0,Y 323.873,Z 374.234,A -85,B 0,C 180,E1 -15969.128,E2 -15969.128} C_VEL
LIN {X 0,Y 322.427,Z 370.116,A -85,B 0,C 180,E1 -15970.28,E2 -15970.28} C_VEL
LIN {X 0,Y 321.635,Z 368.166,A -85,B 0,C 180,E1 -15970.96,E2 -15970.96} C_VEL
LIN {X 0,Y 318.263,Z 362.285,A -85,B 0,C 180,E1 -15974.209,E2 -15974.209} C_VEL
LIN {X 0,Y 316.996,Z 359.025,A -85,B 0,C 180,E1 -15977.024,E2 -15977.024} C_VEL
LIN {X 0,Y 316.904,Z 358.003,A -85,B 0,C 180,E1 -15978.94,E2 -15978.94} C_VEL
LIN {X 0,Y 317.976,Z 357.532,A -85,B 0,C 180,E1 -15981.767,E2 -15981.767} C_VEL
LIN {X 0,Y 318.472,Z 357.86,A -85,B 0,C 180,E1 -15982.603,E2 -15982.603} C_VEL
LIN {X 0,Y 320.621,Z 360.447,A -85,B 0,C 180,E1 -15985.256,E2 -15985.256} C_VEL
LIN {X 0,Y 322.471,Z 363.059,A -85,B 0,C 180,E1 -15986.985,E2 -15986.985} C_VEL
LIN {X 0,Y 325.788,Z 368.686,A -85,B 0,C 180,E1 -15989.644,E2 -15989.644} C_VEL
LIN {X 0,Y 328.835,Z 375.167,A -85,B 0,C 180,E1 -15991.953,E2 -15991.953} C_VEL
LIN {X 0,Y 330.751,Z 380.242,A -85,B 0,C 180,E1 -15993.499,E2 -15993.499} C_VEL
LIN {X 0,Y 331.909,Z 384.572,A -85,B 0,C 180,E1 -15994.648,E2 -15994.648} C_VEL
LIN {X 0,Y 331.962,Z 386.039,A -85,B 0,C 180,E1 -15994.949,E2 -15994.949} C_VEL
LIN {X 0,Y 328.144,Z 397.998,A -85,B 0,C 180,E1 -15996.658,E2 -15996.658} C_VEL
LIN {X 0,Y 324.288,Z 409.302,A -85,B 0,C 180,E1 -15998.708,E2 -15998.708} C_VEL
LIN {X 0,Y 321.252,Z 417.388,A -85,B 0,C 180,E1 -16000.508,E2 -16000.508} C_VEL
LIN {X 0,Y 318.033,Z 425.281,A -85,B 0,C 180,E1 -16002.643,E2 -16002.643} C_VEL
LIN {X 0,Y 315.678,Z 430.732,A -85,B 0,C 180,E1 -16004.505,E2 -16004.505} C_VEL
LIN {X 0,Y 312.889,Z 436.476,A -85,B 0,C 180,E1 -16007.02,E2 -16007.02} C_VEL
LIN {X 0,Y 310.616,Z 440.6,A -85,B 0,C 180,E1 -16009.572,E2 -16009.572} C_VEL
LIN {X 0,Y 308.804,Z 443.147,A -85,B 0,C 180,E1 -16012.152,E2 -16012.152} C_VEL
LIN {X 0,Y 307.632,Z 444.167,A -85,B 0,C 180,E1 -16014.757,E2 -16014.757} C_VEL
LIN {X 0,Y 307.123,Z 444.14,A -85,B 0,C 180,E1 -16016.064,E2 -16016.064} C_VEL
LIN {X 0,Y 306.58,Z 443.757,A -85,B 0,C 180,E1 -16017.372,E2 -16017.372} C_VEL
LIN {X 0,Y 306.323,Z 442.934,A -85,B 0,C 180,E1 -16018.685,E2 -16018.685} C_VEL
LIN {X 0,Y 305.874,Z 441.763,A -85,B 0,C 180,E1 -16020,E2 -16020} C_VEL
LIN {X 0,Y 305.843,Z 440.16,A -85,B 0,C 180,E1 -16021.317,E2 -16021.317} C_VEL
LIN {X 0,Y 305.561,Z 437.03,A -85,B 0,C 180,E1 -16023.297,E2 -16023.297} C_VEL
LIN {X 0,Y 305.728,Z 432.915,A -85,B 0,C 180,E1 -16025.276,E2 -16025.276} C_VEL
LIN {X 0,Y 306.167,Z 427.749,A -85,B 0,C 180,E1 -16027.253,E2 -16027.253} C_VEL
LIN {X 0,Y 306.615,Z 420.724,A -85,B 0,C 180,E1 -16029.433,E2 -16029.433} C_VEL
LIN {X 0,Y 307.295,Z 412.387,A -85,B 0,C 180,E1 -16031.544,E2 -16031.544} C_VEL
LIN {X 0,Y 308.078,Z 402.859,A -85,B 0,C 180,E1 -16033.523,E2 -16033.523} C_VEL
LIN {X 0,Y 309.146,Z 391.353,A -85,B 0,C 180,E1 -16035.493,E2 -16035.493} C_VEL
LIN {X 0,Y 310.276,Z 379.678,A -85,B 0,C 180,E1 -16037.125,E2 -16037.125} C_VEL
LIN {X 0,Y 311.311,Z 367.112,A -85,B 0,C 180,E1 -16038.578,E2 -16038.578} C_VEL
LIN {X 0,Y 312.258,Z 353.661,A -85,B 0,C 180,E1 -16039.827,E2 -16039.827} C_VEL
LIN {X 0,Y 308.868,Z 339.012,A -85,B 0,C 180,E1 -16041.105,E2 -16041.105} C_VEL
LIN {X 0,Y 305.124,Z 324.145,A -85,B 0,C 180,E1 -16042.13,E2 -16042.13} C_VEL
LIN {X 0,Y 304.968,Z 323.288,A -85,B 0,C 180,E1 -16042.187,E2 -16042.187} C_VEL
LIN {X 0,Y 304.951,Z 319.369,A -85,B 0,C 180,E1 -16045.998,E2 -16045.998} C_VEL
LIN {X 0,Y 305.028,Z 316.428,A -85,B 0,C 180,E1 -16048.937,E2 -16048.937} C_VEL
LIN {X 0,Y 304.996,Z 313.455,A -85,B 0,C 180,E1 -16052.005,E2 -16052.005} C_VEL
LIN {X 0,Y 305.19,Z 313.087,A -85,B 0,C 180,E1 -16054.001,E2 -16054.001} C_VEL
LIN {X 0,Y 305.397,Z 313.069,A -85,B 0,C 180,E1 -16056.751,E2 -16056.751} C_VEL
LIN {X 0,Y 305.483,Z 313.26,A -85,B 0,C 180,E1 -16059.037,E2 -16059.037} C_VEL
LIN {X 0,Y 306.084,Z 316.259,A -85,B 0,C 180,E1 -16061.749,E2 -16061.749} C_VEL
LIN {X 0,Y 306.782,Z 320.174,A -85,B 0,C 180,E1 -16065.249,E2 -16065.249} C_VEL
LIN {X 0,Y 307.205,Z 323.898,A -85,B 0,C 180,E1 -16068.437,E2 -16068.437} C_VEL
LIN {X 0,Y 307.209,Z 328.224,A -85,B 0,C 180,E1 -16071.853,E2 -16071.853} C_VEL
LIN {X 0,Y 307.16,Z 333.519,A -85,B 0,C 180,E1 -16075.764,E2 -16075.764} C_VEL
LIN {X 0,Y 308.552,Z 336.808,A -85,B 0,C 180,E1 -16076.047,E2 -16076.047} C_VEL
LIN {X 0,Y 314.97,Z 350.468,A -85,B 0,C 180,E1 -16077.348,E2 -16077.348} C_VEL
LIN {X 0,Y 320.223,Z 364.158,A -85,B 0,C 180,E1 -16078.712,E2 -16078.712} C_VEL
LIN {X 0,Y 324.218,Z 377.409,A -85,B 0,C 180,E1 -16080.12,E2 -16080.12} C_VEL
LIN {X 0,Y 324.952,Z 380.289,A -85,B 0,C 180,E1 -16080.439,E2 -16080.439} C_VEL
LIN {X 0,Y 323.308,Z 394.179,A -85,B 0,C 180,E1 -16081.607,E2 -16081.607} C_VEL
LIN {X 0,Y 321.159,Z 407.59,A -85,B 0,C 180,E1 -16082.994,E2 -16082.994} C_VEL
LIN {X 0,Y 318.783,Z 419.835,A -85,B 0,C 180,E1 -16084.539,E2 -16084.539} C_VEL
LIN {X 0,Y 316.763,Z 430.108,A -85,B 0,C 180,E1 -16086.114,E2 -16086.114} C_VEL
LIN {X 0,Y 314.484,Z 440.566,A -85,B 0,C 180,E1 -16088.017,E2 -16088.017} C_VEL
LIN {X 0,Y 312.417,Z 449.422,A -85,B 0,C 180,E1 -16089.936,E2 -16089.936} C_VEL
LIN {X 0,Y 310.204,Z 458.436,A -85,B 0,C 180,E1 -16092.298,E2 -16092.298} C_VEL
LIN {X 0,Y 308.399,Z 466.174,A -85,B 0,C 180,E1 -16094.807,E2 -16094.807} C_VEL
LIN {X 0,Y 306.92,Z 472.635,A -85,B 0,C 180,E1 -16097.435,E2 -16097.435} C_VEL
LIN {X 0,Y 305.777,Z 477.683,A -85,B 0,C 180,E1 -16100.073,E2 -16100.073} C_VEL
LIN {X 0,Y 305.221,Z 480.575,A -85,B 0,C 180,E1 -16102.059,E2 -16102.059} C_VEL
LIN {X 0,Y 304.718,Z 483.414,A -85,B 0,C 180,E1 -16104.706,E2 -16104.706} C_VEL
LIN {X 0,Y 304.463,Z 485.111,A -85,B 0,C 180,E1 -16107.354,E2 -16107.354} C_VEL
LIN {X 0,Y 304.287,Z 485.707,A -85,B 0,C 180,E1 -16110,E2 -16110} C_VEL
LIN {X 0,Y 304.458,Z 485.147,A -85,B 0,C 180,E1 -16112.646,E2 -16112.646} C_VEL
LIN {X 0,Y 304.7,Z 483.5,A -85,B 0,C 180,E1 -16115.293,E2 -16115.293} C_VEL
LIN {X 0,Y 305.254,Z 480.503,A -85,B 0,C 180,E1 -16118.105,E2 -16118.105} C_VEL
LIN {X 0,Y 306.03,Z 476.722,A -85,B 0,C 180,E1 -16120.586,E2 -16120.586} C_VEL
LIN {X 0,Y 307.224,Z 471.405,A -85,B 0,C 180,E1 -16123.224,E2 -16123.224} C_VEL
LIN {X 0,Y 308.772,Z 464.617,A -85,B 0,C 180,E1 -16125.851,E2 -16125.851} C_VEL
LIN {X 0,Y 310.387,Z 457.77,A -85,B 0,C 180,E1 -16128.011,E2 -16128.011} C_VEL
LIN {X 0,Y 312.651,Z 448.525,A -85,B 0,C 180,E1 -16130.39,E2 -16130.39} C_VEL
LIN {X 0,Y 315.144,Z 437.857,A -85,B 0,C 180,E1 -16132.624,E2 -16132.624} C_VEL
LIN {X 0,Y 317.313,Z 427.071,A -85,B 0,C 180,E1 -16134.508,E2 -16134.508} C_VEL
LIN {X 0,Y 319.867,Z 414.818,A -85,B 0,C 180,E1 -16136.243,E2 -16136.243} C_VEL
LIN {X 0,Y 322.202,Z 401.466,A -85,B 0,C 180,E1 -16137.79,E2 -16137.79} C_VEL
LIN {X 0,Y 324.126,Z 388.494,A -85,B 0,C 180,E1 -16139.012,E2 -16139.012} C_VEL
LIN {X 0,Y 324.967,Z 380.445,A -85,B 0,C 180,E1 -16139.661,E2 -16139.661} C_VEL
LIN {X 0,Y 321.651,Z 368.429,A -85,B 0,C 180,E1 -16140.965,E2 -16140.965} C_VEL
LIN {X 0,Y 317.046,Z 355.333,A -85,B 0,C 180,E1 -16142.287,E2 -16142.287} C_VEL
LIN {X 0,Y 311.539,Z 342.898,A -85,B 0,C 180,E1 -16143.497,E2 -16143.497} C_VEL
LIN {X 0,Y 307.286,Z 334.045,A -85,B 0,C 180,E1 -16144.313,E2 -16144.313} C_VEL
LIN {X 0,Y 307.174,Z 333.5,A -85,B 0,C 180,E1 -16144.391,E2 -16144.391} C_VEL
LIN {X 0,Y 307.215,Z 328.43,A -85,B 0,C 180,E1 -16148.146,E2 -16148.146} C_VEL
LIN {X 0,Y 307.2,Z 324.076,A -85,B 0,C 180,E1 -16151.563,E2 -16151.563} C_VEL
LIN {X 0,Y 306.675,Z 319.757,A -85,B 0,C 180,E1 -16155.269,E2 -16155.269} C_VEL
LIN {X 0,Y 305.916,Z 315.26,A -85,B 0,C 180,E1 -16159.299,E2 -16159.299} C_VEL
LIN {X 0,Y 305.485,Z 313.054,A -85,B 0,C 180,E1 -16161.463,E2 -16161.463} C_VEL
LIN {X 0,Y 305.462,Z 313.063,A -85,B 0,C 180,E1 -16164.887,E2 -16164.887} C_VEL
LIN {X 0,Y 305.441,Z 313.065,A -85,B 0,C 180,E1 -16168.358,E2 -16168.358} C_VEL
LIN {X 0,Y 305.474,Z 313.054,A -85,B 0,C 180,E1 -16171.109,E2 -16171.109} C_VEL
LIN {X 0,Y 305.45,Z 313.049,A -85,B 0,C 180,E1 -16173.467,E2 -16173.467} C_VEL
LIN {X 0,Y 304.815,Z 313.13,A -85,B 0,C 180,E1 -16174.567,E2 -16174.567} C_VEL
LIN {X 0,Y 301.971,Z 313.497,A -85,B 0,C 180,E1 -16176.359,E2 -16176.359} C_VEL
LIN {X 0,Y 299.544,Z 313.79,A -85,B 0,C 180,E1 -16177.812,E2 -16177.812} C_VEL
LIN {X 0,Y 298.509,Z 313.914,A -85,B 0,C 180,E1 -16178.938,E2 -16178.938} C_VEL
LIN {X 0,Y 298.43,Z 313.925,A -85,B 0,C 180,E1 -16179.319,E2 -16179.319} C_VEL
LIN {X 0,Y 298.506,Z 313.913,A -85,B 0,C 180,E1 -16182.177,E2 -16182.177} C_VEL
LIN {X 0,Y 298.585,Z 313.914,A -85,B 0,C 180,E1 -16184.994,E2 -16184.994} C_VEL
LIN {X 0,Y 298.583,Z 313.899,A -85,B 0,C 180,E1 -16189.146,E2 -16189.146} C_VEL
LIN {X 0,Y 298.698,Z 313.9,A -85,B 0,C 180,E1 -16191.884,E2 -16191.884} C_VEL
LIN {X 0,Y 298.637,Z 313.89,A -85,B 0,C 180,E1 -16194.598,E2 -16194.598} C_VEL
LIN {X 0,Y 298.923,Z 313.856,A -85,B 0,C 180,E1 -16198.653,E2 -16198.653} C_VEL
LIN {X 0,Y 298.92,Z 313.867,A -85,B 0,C 180,E1 -16201.347,E2 -16201.347} C_VEL
LIN {X 0,Y 298.753,Z 313.884,A -85,B 0,C 180,E1 -16206.755,E2 -16206.755} C_VEL
LIN {X 0,Y 298.625,Z 313.901,A -85,B 0,C 180,E1 -16209.482,E2 -16209.482} C_VEL
LIN {X 0,Y 298.552,Z 313.923,A -85,B 0,C 180,E1 -16213.615,E2 -16213.615} C_VEL
LIN {X 0,Y 298.548,Z 313.9,A -85,B 0,C 180,E1 -16216.409,E2 -16216.409} C_VEL
LIN {X 0,Y 298.509,Z 313.926,A -85,B 0,C 180,E1 -16219.654,E2 -16219.654} C_VEL
LIN {X 0,Y 298.422,Z 313.936,A -85,B 0,C 180,E1 -16223.6,E2 -16223.6} C_VEL
LIN {X 0,Y 298.407,Z 313.921,A -85,B 0,C 180,E1 -16226.582,E2 -16226.582} C_VEL
LIN {X 0,Y 298.393,Z 313.942,A -85,B 0,C 180,E1 -16229.644,E2 -16229.644} C_VEL
LIN {X 0,Y 298.435,Z 314.008,A -85,B 0,C 180,E1 -16233.601,E2 -16233.601} C_VEL
LIN {X 0,Y 300.145,Z 321.582,A -85,B 0,C 180,E1 -16237.503,E2 -16237.503} C_VEL
LIN {X 0,Y 301.944,Z 329.498,A -85,B 0,C 180,E1 -16241.314,E2 -16241.314} C_VEL
LIN {X 0,Y 304.233,Z 339.389,A -85,B 0,C 180,E1 -16245.735,E2 -16245.735} C_VEL
LIN {X 0,Y 306.435,Z 348.786,A -85,B 0,C 180,E1 -16249.662,E2 -16249.662} C_VEL
LIN {X 0,Y 307.614,Z 354.48,A -85,B 0,C 180,E1 -16251.913,E2 -16251.913} C_VEL
LIN {X 0,Y 306.38,Z 359.887,A -85,B 0,C 180,E1 -16253.795,E2 -16253.795} C_VEL
LIN {X 0,Y 305.984,Z 369.901,A -85,B 0,C 180,E1 -16255.597,E2 -16255.597} C_VEL
LIN {X 0,Y 309.989,Z 388.317,A -85,B 0,C 180,E1 -16256.622,E2 -16256.622} C_VEL
LIN {X 0,Y 312.323,Z 403.948,A -85,B 0,C 180,E1 -16257.584,E2 -16257.584} C_VEL
LIN {X 0,Y 313.625,Z 418.482,A -85,B 0,C 180,E1 -16258.643,E2 -16258.643} C_VEL
LIN {X 0,Y 314.322,Z 433.805,A -85,B 0,C 180,E1 -16259.981,E2 -16259.981} C_VEL
LIN {X 0,Y 313.76,Z 442.05,A -85,B 0,C 180,E1 -16260.745,E2 -16260.745} C_VEL
LIN {X 0,Y 311.37,Z 455.247,A -85,B 0,C 180,E1 -16262.073,E2 -16262.073} C_VEL
LIN {X 0,Y 308.734,Z 467.98,A -85,B 0,C 180,E1 -16263.648,E2 -16263.648} C_VEL
LIN {X 0,Y 306.353,Z 478.682,A -85,B 0,C 180,E1 -16265.25,E2 -16265.25} C_VEL
LIN {X 0,Y 304.014,Z 489.596,A -85,B 0,C 180,E1 -16267.219,E2 -16267.219} C_VEL
LIN {X 0,Y 301.984,Z 498.859,A -85,B 0,C 180,E1 -16269.212,E2 -16269.212} C_VEL
LIN {X 0,Y 300.065,Z 507.955,A -85,B 0,C 180,E1 -16271.567,E2 -16271.567} C_VEL
LIN {X 0,Y 298.517,Z 516.495,A -85,B 0,C 180,E1 -16274.292,E2 -16274.292} C_VEL
LIN {X 0,Y 297.474,Z 523.37,A -85,B 0,C 180,E1 -16277.03,E2 -16277.03} C_VEL
LIN {X 0,Y 296.989,Z 528.774,A -85,B 0,C 180,E1 -16279.777,E2 -16279.777} C_VEL
LIN {X 0,Y 296.912,Z 531.9,A -85,B 0,C 180,E1 -16281.835,E2 -16281.835} C_VEL
LIN {X 0,Y 297.064,Z 534.98,A -85,B 0,C 180,E1 -16284.57,E2 -16284.57} C_VEL
LIN {X 0,Y 297.238,Z 536.824,A -85,B 0,C 180,E1 -16287.29,E2 -16287.29} C_VEL
LIN {X 0,Y 297.346,Z 537.456,A -85,B 0,C 180,E1 -16290,E2 -16290} C_VEL
LIN {X 0,Y 297.276,Z 536.824,A -85,B 0,C 180,E1 -16292.71,E2 -16292.71} C_VEL
LIN {X 0,Y 297.085,Z 534.971,A -85,B 0,C 180,E1 -16295.43,E2 -16295.43} C_VEL
LIN {X 0,Y 296.958,Z 531.88,A -85,B 0,C 180,E1 -16298.164,E2 -16298.164} C_VEL
LIN {X 0,Y 297.085,Z 527.498,A -85,B 0,C 180,E1 -16300.909,E2 -16300.909} C_VEL
LIN {X 0,Y 297.708,Z 521.743,A -85,B 0,C 180,E1 -16303.655,E2 -16303.655} C_VEL
LIN {X 0,Y 298.867,Z 514.461,A -85,B 0,C 180,E1 -16306.391,E2 -16306.391} C_VEL
LIN {X 0,Y 300.312,Z 506.676,A -85,B 0,C 180,E1 -16308.771,E2 -16308.771} C_VEL
LIN {X 0,Y 302.401,Z 497.341,A -85,B 0,C 180,E1 -16311.115,E2 -16311.115} C_VEL
LIN {X 0,Y 304.38,Z 487.842,A -85,B 0,C 180,E1 -16313.112,E2 -16313.112} C_VEL
LIN {X 0,Y 307.082,Z 475.561,A -85,B 0,C 180,E1 -16315.231,E2 -16315.231} C_VEL
LIN {X 0,Y 308.26,Z 470.987,A -85,B 0,C 180,E1 -16316.033,E2 -16316.033} C_VEL
LIN {X 0,Y 312.335,Z 458.382,A -85,B 0,C 180,E1 -16318.199,E2 -16318.199} C_VEL
LIN {X 0,Y 316.563,Z 445.293,A -85,B 0,C 180,E1 -16320.057,E2 -16320.057} C_VEL
LIN {X 0,Y 318.39,Z 437.769,A -85,B 0,C 180,E1 -16321.063,E2 -16321.063} C_VEL
LIN {X 0,Y 320.724,Z 424.498,A -85,B 0,C 180,E1 -16322.778,E2 -16322.778} C_VEL
LIN {X 0,Y 321.703,Z 413.567,A -85,B 0,C 180,E1 -16324.232,E2 -16324.232} C_VEL
LIN {X 0,Y 321.73,Z 400.764,A -85,B 0,C 180,E1 -16326.076,E2 -16326.076} C_VEL
LIN {X 0,Y 321.106,Z 388.825,A -85,B 0,C 180,E1 -16328.008,E2 -16328.008} C_VEL
LIN {X 0,Y 320.218,Z 379.086,A -85,B 0,C 180,E1 -16329.811,E2 -16329.811} C_VEL
LIN {X 0,Y 318.984,Z 375.181,A -85,B 0,C 180,E1 -16331.008,E2 -16331.008} C_VEL
LIN {X 0,Y 318.477,Z 374.046,A -85,B 0,C 180,E1 -16331.455,E2 -16331.455} C_VEL
LIN {X 0,Y 316.392,Z 370.301,A -85,B 0,C 180,E1 -16333.52,E2 -16333.52} C_VEL
LIN {X 0,Y 315.1,Z 367.357,A -85,B 0,C 180,E1 -16335.54,E2 -16335.54} C_VEL
LIN {X 0,Y 314.494,Z 365.196,A -85,B 0,C 180,E1 -16337.901,E2 -16337.901} C_VEL
LIN {X 0,Y 314.55,Z 364.484,A -85,B 0,C 180,E1 -16339.613,E2 -16339.613} C_VEL
LIN {X 0,Y 315.156,Z 364.165,A -85,B 0,C 180,E1 -16341.362,E2 -16341.362} C_VEL
LIN {X 0,Y 316.106,Z 365.126,A -85,B 0,C 180,E1 -16343.168,E2 -16343.168} C_VEL
LIN {X 0,Y 317.486,Z 366.719,A -85,B 0,C 180,E1 -16344.99,E2 -16344.99} C_VEL
LIN {X 0,Y 319.155,Z 369.243,A -85,B 0,C 180,E1 -16346.803,E2 -16346.803} C_VEL
LIN {X 0,Y 321.827,Z 374.274,A -85,B 0,C 180,E1 -16349.317,E2 -16349.317} C_VEL
LIN {X 0,Y 324.733,Z 381.272,A -85,B 0,C 180,E1 -16351.95,E2 -16351.95} C_VEL
LIN {X 0,Y 326.558,Z 387.652,A -85,B 0,C 180,E1 -16353.9,E2 -16353.9} C_VEL
LIN {X 0,Y 326.754,Z 388.829,A -85,B 0,C 180,E1 -16354.219,E2 -16354.219} C_VEL
LIN {X 0,Y 322.889,Z 400.188,A -85,B 0,C 180,E1 -16355.914,E2 -16355.914} C_VEL
LIN {X 0,Y 319.368,Z 409.794,A -85,B 0,C 180,E1 -16357.691,E2 -16357.691} C_VEL
LIN {X 0,Y 315.559,Z 419.16,A -85,B 0,C 180,E1 -16359.806,E2 -16359.806} C_VEL
LIN {X 0,Y 312.599,Z 425.841,A -85,B 0,C 180,E1 -16361.654,E2 -16361.654} C_VEL
LIN {X 0,Y 309.954,Z 431.403,A -85,B 0,C 180,E1 -16363.535,E2 -16363.535} C_VEL
LIN {X 0,Y 307.623,Z 435.972,A -85,B 0,C 180,E1 -16365.445,E2 -16365.445} C_VEL
LIN {X 0,Y 305,Z 440.616,A -85,B 0,C 180,E1 -16368.031,E2 -16368.031} C_VEL
LIN {X 0,Y 302.81,Z 443.69,A -85,B 0,C 180,E1 -16370.65,E2 -16370.65} C_VEL
LIN {X 0,Y 301.234,Z 445.246,A -85,B 0,C 180,E1 -16373.301,E2 -16373.301} C_VEL
LIN {X 0,Y 300.684,Z 445.484,A -85,B 0,C 180,E1 -16374.636,E2 -16374.636} C_VEL
LIN {X 0,Y 300.156,Z 445.349,A -85,B 0,C 180,E1 -16375.972,E2 -16375.972} C_VEL
LIN {X 0,Y 299.579,Z 444.839,A -85,B 0,C 180,E1 -16377.311,E2 -16377.311} C_VEL
LIN {X 0,Y 299.308,Z 443.919,A -85,B 0,C 180,E1 -16378.655,E2 -16378.655} C_VEL
LIN {X 0,Y 298.845,Z 442.661,A -85,B 0,C 180,E1 -16380,E2 -16380} C_VEL
LIN {X 0,Y 298.697,Z 439.972,A -85,B 0,C 180,E1 -16382.023,E2 -16382.023} C_VEL
LIN {X 0,Y 298.438,Z 436.382,A -85,B 0,C 180,E1 -16384.051,E2 -16384.051} C_VEL
LIN {X 0,Y 298.868,Z 431.757,A -85,B 0,C 180,E1 -16386.075,E2 -16386.075} C_VEL
LIN {X 0,Y 299.302,Z 425.015,A -85,B 0,C 180,E1 -16388.439,E2 -16388.439} C_VEL
LIN {X 0,Y 299.976,Z 416.59,A -85,B 0,C 180,E1 -16390.803,E2 -16390.803} C_VEL
LIN {X 0,Y 300.738,Z 407.698,A -85,B 0,C 180,E1 -16392.827,E2 -16392.827} C_VEL
LIN {X 0,Y 301.631,Z 397,A -85,B 0,C 180,E1 -16394.851,E2 -16394.851} C_VEL
LIN {X 0,Y 302.838,Z 385.072,A -85,B 0,C 180,E1 -16396.69,E2 -16396.69} C_VEL
LIN {X 0,Y 303.964,Z 372.622,A -85,B 0,C 180,E1 -16398.273,E2 -16398.273} C_VEL
LIN {X 0,Y 305.061,Z 358.809,A -85,B 0,C 180,E1 -16399.69,E2 -16399.69} C_VEL
LIN {X 0,Y 305.356,Z 355.106,A -85,B 0,C 180,E1 -16400.021,E2 -16400.021} C_VEL
LIN {X 0,Y 301.888,Z 339.98,A -85,B 0,C 180,E1 -16401.375,E2 -16401.375} C_VEL
LIN {X 0,Y 298.035,Z 324.61,A -85,B 0,C 180,E1 -16402.47,E2 -16402.47} C_VEL
LIN {X 0,Y 297.912,Z 323.853,A -85,B 0,C 180,E1 -16402.559,E2 -16402.559} C_VEL
LIN {X 0,Y 297.91,Z 319.709,A -85,B 0,C 180,E1 -16406.63,E2 -16406.63} C_VEL
LIN {X 0,Y 297.97,Z 316.69,A -85,B 0,C 180,E1 -16409.69,E2 -16409.69} C_VEL
LIN {X 0,Y 297.962,Z 313.997,A -85,B 0,C 180,E1 -16412.58,E2 -16412.58} C_VEL
LIN {X 0,Y 298.311,Z 313.951,A -85,B 0,C 180,E1 -16416.085,E2 -16416.085} C_VEL
LIN {X 0,Y 298.386,Z 314.089,A -85,B 0,C 180,E1 -16417.929,E2 -16417.929} C_VEL
LIN {X 0,Y 299.182,Z 317.693,A -85,B 0,C 180,E1 -16421.261,E2 -16421.261} C_VEL
LIN {X 0,Y 299.961,Z 322.187,A -85,B 0,C 180,E1 -16425.34,E2 -16425.34} C_VEL
LIN {X 0,Y 300.356,Z 325.838,A -85,B 0,C 180,E1 -16428.484,E2 -16428.484} C_VEL
LIN {X 0,Y 300.349,Z 329.871,A -85,B 0,C 180,E1 -16431.677,E2 -16431.677} C_VEL
LIN {X 0,Y 300.347,Z 334.187,A -85,B 0,C 180,E1 -16434.889,E2 -16434.889} C_VEL
LIN {X 0,Y 301.706,Z 337.365,A -85,B 0,C 180,E1 -16435.165,E2 -16435.165} C_VEL
LIN {X 0,Y 308.443,Z 351.587,A -85,B 0,C 180,E1 -16436.591,E2 -16436.591} C_VEL
LIN {X 0,Y 313.409,Z 364.414,A -85,B 0,C 180,E1 -16437.926,E2 -16437.926} C_VEL
LIN {X 0,Y 317.515,Z 377.741,A -85,B 0,C 180,E1 -16439.396,E2 -16439.396} C_VEL
LIN {X 0,Y 318.721,Z 382.657,A -85,B 0,C 180,E1 -16439.955,E2 -16439.955} C_VEL
LIN {X 0,Y 316.852,Z 396.466,A -85,B 0,C 180,E1 -16441.155,E2 -16441.155} C_VEL
LIN {X 0,Y 314.639,Z 409.564,A -85,B 0,C 180,E1 -16442.568,E2 -16442.568} C_VEL
LIN {X 0,Y 312.313,Z 420.888,A -85,B 0,C 180,E1 -16444.043,E2 -16444.043} C_VEL
LIN {X 0,Y 309.872,Z 432.61,A -85,B 0,C 180,E1 -16445.905,E2 -16445.905} C_VEL
LIN {X 0,Y 307.508,Z 442.756,A -85,B 0,C 180,E1 -16447.845,E2 -16447.845} C_VEL
LIN {X 0,Y 305.077,Z 452.659,A -85,B 0,C 180,E1 -16450.135,E2 -16450.135} C_VEL
LIN {X 0,Y 303.021,Z 460.863,A -85,B 0,C 180,E1 -16452.451,E2 -16452.451} C_VEL
LIN {X 0,Y 301.136,Z 468.53,A -85,B 0,C 180,E1 -16455.124,E2 -16455.124} C_VEL
LIN {X 0,Y 299.691,Z 474.615,A -85,B 0,C 180,E1 -16457.815,E2 -16457.815} C_VEL
LIN {X 0,Y 298.593,Z 479.315,A -85,B 0,C 180,E1 -16460.516,E2 -16460.516} C_VEL
LIN {X 0,Y 297.806,Z 482.759,A -85,B 0,C 180,E1 -16463.223,E2 -16463.223} C_VEL
LIN {X 0,Y 297.593,Z 485.003,A -85,B 0,C 180,E1 -16465.937,E2 -16465.937} C_VEL
LIN {X 0,Y 297.266,Z 486.162,A -85,B 0,C 180,E1 -16468.645,E2 -16468.645} C_VEL
LIN {X 0,Y 297.265,Z 486.174,A -85,B 0,C 180,E1 -16471.354,E2 -16471.354} C_VEL
LIN {X 0,Y 297.581,Z 485.063,A -85,B 0,C 180,E1 -16474.063,E2 -16474.063} C_VEL
LIN {X 0,Y 297.805,Z 482.868,A -85,B 0,C 180,E1 -16476.776,E2 -16476.776} C_VEL
LIN {X 0,Y 298.59,Z 479.484,A -85,B 0,C 180,E1 -16479.483,E2 -16479.483} C_VEL
LIN {X 0,Y 299.629,Z 474.846,A -85,B 0,C 180,E1 -16482.187,E2 -16482.187} C_VEL
LIN {X 0,Y 301.089,Z 468.813,A -85,B 0,C 180,E1 -16484.878,E2 -16484.878} C_VEL
LIN {X 0,Y 302.961,Z 461.21,A -85,B 0,C 180,E1 -16487.552,E2 -16487.552} C_VEL
LIN {X 0,Y 304.988,Z 453.087,A -85,B 0,C 180,E1 -16489.87,E2 -16489.87} C_VEL
LIN {X 0,Y 307.457,Z 443.264,A -85,B 0,C 180,E1 -16492.158,E2 -16492.158} C_VEL
LIN {X 0,Y 309.779,Z 433.222,A -85,B 0,C 180,E1 -16494.102,E2 -16494.102} C_VEL
LIN {X 0,Y 311.97,Z 422.934,A -85,B 0,C 180,E1 -16495.769,E2 -16495.769} C_VEL
LIN {X 0,Y 314.531,Z 410.389,A -85,B 0,C 180,E1 -16497.442,E2 -16497.442} C_VEL
LIN {X 0,Y 316.721,Z 397.449,A -85,B 0,C 180,E1 -16498.857,E2 -16498.857} C_VEL
LIN {X 0,Y 318.69,Z 383.456,A -85,B 0,C 180,E1 -16500.088,E2 -16500.088} C_VEL
LIN {X 0,Y 318.461,Z 381.45,A -85,B 0,C 180,E1 -16500.296,E2 -16500.296} C_VEL
LIN {X 0,Y 315.175,Z 369.562,A -85,B 0,C 180,E1 -16501.634,E2 -16501.634} C_VEL
LIN {X 0,Y 310.7,Z 356.878,A -85,B 0,C 180,E1 -16502.975,E2 -16502.975} C_VEL
LIN {X 0,Y 305.11,Z 344.223,A -85,B 0,C 180,E1 -16504.271,E2 -16504.271} C_VEL
LIN {X 0,Y 300.433,Z 334.565,A -85,B 0,C 180,E1 -16505.211,E2 -16505.211} C_VEL
LIN {X 0,Y 300.354,Z 334.122,A -85,B 0,C 180,E1 -16505.286,E2 -16505.286} C_VEL
LIN {X 0,Y 300.352,Z 328.583,A -85,B 0,C 180,E1 -16509.45,E2 -16509.45} C_VEL
LIN {X 0,Y 300.218,Z 324.52,A -85,B 0,C 180,E1 -16512.756,E2 -16512.756} C_VEL
LIN {X 0,Y 299.827,Z 321.614,A -85,B 0,C 180,E1 -16515.315,E2 -16515.315} C_VEL
LIN {X 0,Y 299.162,Z 317.705,A -85,B 0,C 180,E1 -16518.869,E2 -16518.869} C_VEL
LIN {X 0,Y 298.437,Z 313.934,A -85,B 0,C 180,E1 -16522.512,E2 -16522.512} C_VEL
LIN {X 0,Y 298.408,Z 313.935,A -85,B 0,C 180,E1 -16525.581,E2 -16525.581} C_VEL
LIN {X 0,Y 298.377,Z 313.939,A -85,B 0,C 180,E1 -16528.789,E2 -16528.789} C_VEL
LIN {X 0,Y 298.411,Z 313.941,A -85,B 0,C 180,E1 -16531.899,E2 -16531.899} C_VEL
LIN {X 0,Y 298.442,Z 313.926,A -85,B 0,C 180,E1 -16534.92,E2 -16534.92} C_VEL
LIN {X 0,Y 298.412,Z 313.923,A -85,B 0,C 180,E1 -16537.863,E2 -16537.863} C_VEL
LIN {X 0,Y 298.43,Z 313.925,A -85,B 0,C 180,E1 -16539.319,E2 -16539.319} C_VEL
LIN {X 0,Y 297.782,Z 314.018,A -85,B 0,C 180,E1 -16540.447,E2 -16540.447} C_VEL
LIN {X 0,Y 294.965,Z 314.36,A -85,B 0,C 180,E1 -16542.283,E2 -16542.283} C_VEL
LIN {X 0,Y 292.577,Z 314.655,A -85,B 0,C 180,E1 -16543.774,E2 -16543.774} C_VEL
LIN {X 0,Y 291.562,Z 314.788,A -85,B 0,C 180,E1 -16544.928,E2 -16544.928} C_VEL
LIN {X 0,Y 291.485,Z 314.795,A -85,B 0,C 180,E1 -16545.318,E2 -16545.318} C_VEL
LIN {X 0,Y 291.529,Z 314.775,A -85,B 0,C 180,E1 -16548.88,E2 -16548.88} C_VEL
LIN {X 0,Y 291.651,Z 314.779,A -85,B 0,C 180,E1 -16551.687,E2 -16551.687} C_VEL
LIN {X 0,Y 291.606,Z 314.764,A -85,B 0,C 180,E1 -16554.468,E2 -16554.468} C_VEL
LIN {X 0,Y 291.889,Z 314.732,A -85,B 0,C 180,E1 -16558.62,E2 -16558.62} C_VEL
LIN {X 0,Y 291.886,Z 314.743,A -85,B 0,C 180,E1 -16561.38,E2 -16561.38} C_VEL
LIN {X 0,Y 291.704,Z 314.764,A -85,B 0,C 180,E1 -16566.919,E2 -16566.919} C_VEL
LIN {X 0,Y 291.568,Z 314.776,A -85,B 0,C 180,E1 -16569.714,E2 -16569.714} C_VEL
LIN {X 0,Y 291.522,Z 314.797,A -85,B 0,C 180,E1 -16573.95,E2 -16573.95} C_VEL
LIN {X 0,Y 291.486,Z 314.78,A -85,B 0,C 180,E1 -16576.818,E2 -16576.818} C_VEL
LIN {X 0,Y 291.45,Z 314.802,A -85,B 0,C 180,E1 -16579.875,E2 -16579.875} C_VEL
LIN {X 0,Y 291.363,Z 314.818,A -85,B 0,C 180,E1 -16584.208,E2 -16584.208} C_VEL
LIN {X 0,Y 291.353,Z 314.802,A -85,B 0,C 180,E1 -16587.278,E2 -16587.278} C_VEL
LIN {X 0,Y 291.318,Z 314.823,A -85,B 0,C 180,E1 -16590.439,E2 -16590.439} C_VEL
LIN {X 0,Y 291.379,Z 314.859,A -85,B 0,C 180,E1 -16592.892,E2 -16592.892} C_VEL
LIN {X 0,Y 293.008,Z 322.262,A -85,B 0,C 180,E1 -16596.844,E2 -16596.844} C_VEL
LIN {X 0,Y 294.565,Z 329.057,A -85,B 0,C 180,E1 -16600.228,E2 -16600.228} C_VEL
LIN {X 0,Y 296.437,Z 337.347,A -85,B 0,C 180,E1 -16604.111,E2 -16604.111} C_VEL
LIN {X 0,Y 298.473,Z 345.913,A -85,B 0,C 180,E1 -16607.878,E2 -16607.878} C_VEL
LIN {X 0,Y 300.407,Z 354.05,A -85,B 0,C 180,E1 -16611.258,E2 -16611.258} C_VEL
LIN {X 0,Y 300.48,Z 356.245,A -85,B 0,C 180,E1 -16612.123,E2 -16612.123} C_VEL
LIN {X 0,Y 300.227,Z 357.377,A -85,B 0,C 180,E1 -16612.51,E2 -16612.51} C_VEL
LIN {X 0,Y 299.595,Z 369.289,A -85,B 0,C 180,E1 -16614.743,E2 -16614.743} C_VEL
LIN {X 0,Y 304.003,Z 389.604,A -85,B 0,C 180,E1 -16615.937,E2 -16615.937} C_VEL
LIN {X 0,Y 306.242,Z 405.567,A -85,B 0,C 180,E1 -16616.976,E2 -16616.976} C_VEL
LIN {X 0,Y 307.468,Z 421.19,A -85,B 0,C 180,E1 -16618.185,E2 -16618.185} C_VEL
LIN {X 0,Y 307.92,Z 435.413,A -85,B 0,C 180,E1 -16619.5,E2 -16619.5} C_VEL
LIN {X 0,Y 307.306,Z 442.911,A -85,B 0,C 180,E1 -16620.225,E2 -16620.225} C_VEL
LIN {X 0,Y 304.781,Z 456.081,A -85,B 0,C 180,E1 -16621.602,E2 -16621.602} C_VEL
LIN {X 0,Y 302.073,Z 468.558,A -85,B 0,C 180,E1 -16623.207,E2 -16623.207} C_VEL
LIN {X 0,Y 299.835,Z 478.074,A -85,B 0,C 180,E1 -16624.674,E2 -16624.674} C_VEL
LIN {X 0,Y 297.371,Z 488.982,A -85,B 0,C 180,E1 -16626.68,E2 -16626.68} C_VEL
LIN {X 0,Y 294.926,Z 499.621,A -85,B 0,C 180,E1 -16629.057,E2 -16629.057} C_VEL
LIN {X 0,Y 292.986,Z 508.48,A -85,B 0,C 180,E1 -16631.468,E2 -16631.468} C_VEL
LIN {X 0,Y 291.601,Z 515.88,A -85,B 0,C 180,E1 -16633.909,E2 -16633.909} C_VEL
LIN {X 0,Y 290.455,Z 522.752,A -85,B 0,C 180,E1 -16636.711,E2 -16636.711} C_VEL
LIN {X 0,Y 289.934,Z 528.159,A -85,B 0,C 180,E1 -16639.526,E2 -16639.526} C_VEL
LIN {X 0,Y 289.832,Z 531.285,A -85,B 0,C 180,E1 -16641.635,E2 -16641.635} C_VEL
LIN {X 0,Y 289.984,Z 534.369,A -85,B 0,C 180,E1 -16644.437,E2 -16644.437} C_VEL
LIN {X 0,Y 290.154,Z 536.215,A -85,B 0,C 180,E1 -16647.224,E2 -16647.224} C_VEL
LIN {X 0,Y 290.276,Z 536.848,A -85,B 0,C 180,E1 -16650,E2 -16650} C_VEL
LIN {X 0,Y 290.19,Z 536.214,A -85,B 0,C 180,E1 -16652.777,E2 -16652.777} C_VEL
LIN {X 0,Y 290.001,Z 534.359,A -85,B 0,C 180,E1 -16655.563,E2 -16655.563} C_VEL
LIN {X 0,Y 289.875,Z 531.265,A -85,B 0,C 180,E1 -16658.365,E2 -16658.365} C_VEL
LIN {X 0,Y 290.03,Z 526.88,A -85,B 0,C 180,E1 -16661.178,E2 -16661.178} C_VEL
LIN {X 0,Y 290.722,Z 521.125,A -85,B 0,C 180,E1 -16663.99,E2 -16663.99} C_VEL
LIN {X 0,Y 291.927,Z 513.839,A -85,B 0,C 180,E1 -16666.792,E2 -16666.792} C_VEL
LIN {X 0,Y 293.502,Z 506.058,A -85,B 0,C 180,E1 -16669.224,E2 -16669.224} C_VEL
LIN {X 0,Y 295.685,Z 496.781,A -85,B 0,C 180,E1 -16671.605,E2 -16671.605} C_VEL
LIN {X 0,Y 297.789,Z 487.228,A -85,B 0,C 180,E1 -16673.654,E2 -16673.654} C_VEL
LIN {X 0,Y 300.386,Z 476.155,A -85,B 0,C 180,E1 -16675.648,E2 -16675.648} C_VEL
LIN {X 0,Y 304.314,Z 464.821,A -85,B 0,C 180,E1 -16677.883,E2 -16677.883} C_VEL
LIN {X 0,Y 308.892,Z 451.624,A -85,B 0,C 180,E1 -16680.037,E2 -16680.037} C_VEL
LIN {X 0,Y 312.051,Z 441.924,A -85,B 0,C 180,E1 -16681.388,E2 -16681.388} C_VEL
LIN {X 0,Y 315.206,Z 427.074,A -85,B 0,C 180,E1 -16683.444,E2 -16683.444} C_VEL
LIN {X 0,Y 316.533,Z 416.534,A -85,B 0,C 180,E1 -16684.92,E2 -16684.92} C_VEL
LIN {X 0,Y 317.071,Z 402.586,A -85,B 0,C 180,E1 -16687.065,E2 -16687.065} C_VEL
LIN {X 0,Y 316.847,Z 389.693,A -85,B 0,C 180,E1 -16689.316,E2 -16689.316} C_VEL
LIN {X 0,Y 316.547,Z 384.109,A -85,B 0,C 180,E1 -16690.439,E2 -16690.439} C_VEL
LIN {X 0,Y 315.699,Z 381.021,A -85,B 0,C 180,E1 -16691.432,E2 -16691.432} C_VEL
LIN {X 0,Y 314.082,Z 377.797,A -85,B 0,C 180,E1 -16693.075,E2 -16693.075} C_VEL
LIN {X 0,Y 312.378,Z 373.767,A -85,B 0,C 180,E1 -16695.777,E2 -16695.777} C_VEL
LIN {X 0,Y 311.859,Z 371.73,A -85,B 0,C 180,E1 -16698.047,E2 -16698.047} C_VEL
LIN {X 0,Y 312.223,Z 370.796,A -85,B 0,C 180,E1 -16700.93,E2 -16700.93} C_VEL
LIN {X 0,Y 312.921,Z 371.315,A -85,B 0,C 180,E1 -16702.67,E2 -16702.67} C_VEL
LIN {X 0,Y 313.919,Z 372.613,A -85,B 0,C 180,E1 -16704.403,E2 -16704.403} C_VEL
LIN {X 0,Y 315.846,Z 375.776,A -85,B 0,C 180,E1 -16706.863,E2 -16706.863} C_VEL
LIN {X 0,Y 318.208,Z 380.88,A -85,B 0,C 180,E1 -16709.471,E2 -16709.471} C_VEL
LIN {X 0,Y 320.402,Z 387.169,A -85,B 0,C 180,E1 -16711.925,E2 -16711.925} C_VEL
LIN {X 0,Y 321.548,Z 392.333,A -85,B 0,C 180,E1 -16713.568,E2 -16713.568} C_VEL
LIN {X 0,Y 317.091,Z 404.127,A -85,B 0,C 180,E1 -16715.445,E2 -16715.445} C_VEL
LIN {X 0,Y 312.793,Z 414.675,A -85,B 0,C 180,E1 -16717.545,E2 -16717.545} C_VEL
LIN {X 0,Y 309.292,Z 422.436,A -85,B 0,C 180,E1 -16719.463,E2 -16719.463} C_VEL
LIN {X 0,Y 305.343,Z 430.41,A -85,B 0,C 180,E1 -16721.897,E2 -16721.897} C_VEL
LIN {X 0,Y 302.7,Z 435.328,A -85,B 0,C 180,E1 -16723.823,E2 -16723.823} C_VEL
LIN {X 0,Y 300.317,Z 439.364,A -85,B 0,C 180,E1 -16725.776,E2 -16725.776} C_VEL
LIN {X 0,Y 298.31,Z 442.476,A -85,B 0,C 180,E1 -16727.759,E2 -16727.759} C_VEL
LIN {X 0,Y 295.992,Z 445.31,A -85,B 0,C 180,E1 -16730.433,E2 -16730.433} C_VEL
LIN {X 0,Y 294.327,Z 446.671,A -85,B 0,C 180,E1 -16733.143,E2 -16733.143} C_VEL
LIN {X 0,Y 293.184,Z 446.505,A -85,B 0,C 180,E1 -16735.876,E2 -16735.876} C_VEL
LIN {X 0,Y 292.576,Z 445.907,A -85,B 0,C 180,E1 -16737.246,E2 -16737.246} C_VEL
LIN {X 0,Y 292.292,Z 444.896,A -85,B 0,C 180,E1 -16738.622,E2 -16738.622} C_VEL
LIN {X 0,Y 291.816,Z 443.546,A -85,B 0,C 180,E1 -16740,E2 -16740} C_VEL
LIN {X 0,Y 291.635,Z 440.701,A -85,B 0,C 180,E1 -16742.072,E2 -16742.072} C_VEL
LIN {X 0,Y 291.396,Z 436.948,A -85,B 0,C 180,E1 -16744.149,E2 -16744.149} C_VEL
LIN {X 0,Y 291.821,Z 432.159,A -85,B 0,C 180,E1 -16746.222,E2 -16746.222} C_VEL
